// TwinCAT 3 PLC project TwinCAT_OpenFramework_IO_Models
// Title: TwinCAT Open Framework IO Models
// Company: Oleksandr Tiutyk FOP
// Author: Oleksandr Tiutyk
// ProjectVersion: 1.0.13.0
// Description: Beckhoff I/O (input/output) models: different terminal models
// ProgramVersion: 3.1.4026.28
// project tree:
//   AnalogIO/Inputs/ ANALOG_INPUT_DINT_CHANNEL.TcDUT, ANALOG_INPUT_REAL_CHANNEL.TcDUT, ANALOG_INPUT_INT_CHANNEL.TcDUT, RTD_INPUT_CHANNEL.TcDUT, THERMOCOUPLE_INPUT_CHANNEL.TcDUT
//   AnalogIO/Inputs/EL3002/ EL3002.TcDUT, EL3002_EX.TcDUT
//   AnalogIO/Inputs/EL3004/ EL3004.TcDUT, EL3004_EX.TcDUT
//   AnalogIO/Inputs/EL3008/ EL3008.TcDUT, EL3008_EX.TcDUT
//   AnalogIO/Inputs/EL3078/ EL3078.TcDUT, EL3078_EX.TcDUT
//   AnalogIO/Inputs/EL3001/ EL3001.TcDUT, EL3001_EX.TcDUT
//   AnalogIO/Outputs/EL4001/ EL4001.TcDUT, EL4001_EX.TcDUT
//   AnalogIO/Outputs/EL4002/ EL4002.TcDUT, EL4002_EX.TcDUT
//   AnalogIO/Outputs/EL4004/ EL4004.TcDUT, EL4004_EX.TcDUT
//   AnalogIO/Outputs/EL4008/ EL4008.TcDUT, EL4008_EX.TcDUT
//   DigitalIO/Inputs/EL1002/ EL1002.TcDUT, EL1002_EX.TcDUT
//   DigitalIO/Inputs/EL1004/ EL1004.TcDUT, EL1004_EX.TcDUT
//   DigitalIO/Inputs/EL1018/ EL1018_EX.TcDUT, EL1018.TcDUT
//   DigitalIO/Inputs/EL1809/ EL1809.TcDUT, EL1809_EX.TcDUT
//   DigitalIO/Outputs/EL2008/ EL2008.TcDUT, EL2008_EX.TcDUT
//   DigitalIO/Outputs/EL2002/ EL2002.TcDUT, EL2002_EX.TcDUT
//   DigitalIO/Outputs/EL2004/ EL2004.TcDUT, EL2004_EX.TcDUT
//   DigitalIO/Outputs/EL2409/ EL2409.TcDUT, EL2409_EX.TcDUT
//   Internal/ CurrentNamespace.TcPOU, NamespaceExtractor.TcPOU
//   Serial/EL6022/ EL6022.TcDUT, EL6022_CHANNEL.TcDUT, EL6022_EX.TcDUT
//   Serial/ EL6xxx22ByteInData.TcDUT, EL6xxx22ByteOutData.TcDUT
//   AnalogIO/Inputs/EL3201/ EL3201.TcDUT, EL3201_EX.TcDUT
//   AnalogIO/Inputs/EL3202/ EL3202.TcDUT, EL3202_EX.TcDUT
//   AnalogIO/Inputs/EL3204/ EL3204.TcDUT, EL3204_EX.TcDUT
//   AnalogIO/Inputs/EL3208/ EL3208.TcDUT, EL3208_EX.TcDUT
//   AnalogIO/Inputs/EL3311/ EL3311.TcDUT, EL3311_EX.TcDUT
//   AnalogIO/Inputs/EL3312/ EL3312.TcDUT, EL3312_EX.TcDUT
//   AnalogIO/Inputs/EL3314/ EL3314.TcDUT, EL3314_EX.TcDUT
//   AnalogIO/Inputs/EL3318/ EL3318.TcDUT, EL3318_EX.TcDUT
//   DigitalIO/Inputs/EL1008/ EL1008.TcDUT, EL1008_EX.TcDUT
//   DigitalIO/Outputs/EL2809/ EL2809.TcDUT, EL2809_EX.TcDUT
//   DigitalIO/Outputs/EL2622/ EL2622.TcDUT, EL2622_EX.TcDUT
//   DigitalIO/Outputs/EL2624/ EL2624.TcDUT, EL2624_EX.TcDUT
//   Serial/EL6001/ EL6001.TcDUT, EL6001_CHANNEL.TcDUT, EL6001_EX.TcDUT
//   Serial/EL6002/ EL6002.TcDUT, EL6002_CHANNEL.TcDUT, EL6002_EX.TcDUT
//   Serial/EL6021/ EL6021.TcDUT, EL6021_CHANNEL.TcDUT, EL6021_EX.TcDUT
//   Counters/ COUNTER_INPUT_CHANNEL.TcDUT, COUNTER_OUTPUT_CHANNEL.TcDUT, COUNTER_CHANNEL.TcDUT
//   Counters/EL1502/ EL1502.TcDUT, EL1502_EX.TcDUT
//   Counters/EL1512/ EL1512.TcDUT, EL1512_EX.TcDUT
//   Encoders/ INCREMENTAL_ENCODER_INPUT_CHANNEL.TcDUT, INCREMENTAL_ENCODER_OUTPUT_CHANNEL.TcDUT, INCREMENTAL_ENCODER_CHANNEL.TcDUT, INCREMENTAL_ENCODER_COUNTER_INPUT_CHANNEL.TcDUT, INCREMENTAL_ENCODER_COUNTER_CHANNEL.TcDUT, SSI_ENCODER_CHANNEL.TcDUT
//   Encoders/EL5101/ EL5101.TcDUT, EL5101_EX.TcDUT
//   Encoders/EL5151/ EL5151.TcDUT, EL5151_EX.TcDUT
//   Encoders/EL5152/ EL5152.TcDUT, EL5152_EX.TcDUT
//   Encoders/EL5001/ EL5001.TcDUT, EL5001_EX.TcDUT
//   Encoders/EL5002/ EL5002.TcDUT, EL5002_EX.TcDUT
//   PWM/ PWM_OUTPUT_CHANNEL.TcDUT, PULSE_TRAIN_INPUT_CHANNEL.TcDUT, PULSE_TRAIN_OUTPUT_CHANNEL.TcDUT, PULSE_TRAIN_CHANNEL.TcDUT
//   PWM/EL2502/ EL2502.TcDUT, EL2502_EX.TcDUT
//   PWM/EL2521/ EL2521.TcDUT, EL2521_EX.TcDUT
//   Version/ Global_Version.TcGVL
//   AnalogIO/Inputs/EL3051/ EL3051.TcDUT, EL3051_EX.TcDUT
//   AnalogIO/Inputs/EL3052/ EL3052.TcDUT, EL3052_EX.TcDUT
//   AnalogIO/Inputs/EL3054/ EL3054.TcDUT, EL3054_EX.TcDUT
//   AnalogIO/Inputs/EL3058/ EL3058.TcDUT, EL3058_EX.TcDUT
//   AnalogIO/Inputs/EL3102/ EL3102.TcDUT, EL3102_EX.TcDUT
//   AnalogIO/Inputs/EL3104/ EL3104.TcDUT, EL3104_EX.TcDUT
//   AnalogIO/Inputs/EL3122/ EL3122.TcDUT, EL3122_EX.TcDUT
//   AnalogIO/Inputs/EL3124/ EL3124.TcDUT, EL3124_EX.TcDUT
//   AnalogIO/Outputs/EL4021/ EL4021.TcDUT, EL4021_EX.TcDUT
//   AnalogIO/Outputs/EL4022/ EL4022.TcDUT, EL4022_EX.TcDUT
//   AnalogIO/Outputs/EL4024/ EL4024.TcDUT, EL4024_EX.TcDUT
//   AnalogIO/Outputs/EL4028/ EL4028.TcDUT, EL4028_EX.TcDUT
//   AnalogIO/Outputs/EL4102/ EL4102.TcDUT, EL4102_EX.TcDUT
//   AnalogIO/Outputs/EL4104/ EL4104.TcDUT, EL4104_EX.TcDUT
//   AnalogIO/Outputs/EL4132/ EL4132.TcDUT, EL4132_EX.TcDUT
//   AnalogIO/Outputs/EL4134/ EL4134.TcDUT, EL4134_EX.TcDUT
//   AnalogIO/Outputs/EL4122/ EL4122.TcDUT, EL4122_EX.TcDUT
//   AnalogIO/Outputs/EL4124/ EL4124.TcDUT, EL4124_EX.TcDUT
//   Weighing/ STRAIN_GAUGE_INPUT_CHANNEL.TcDUT, STRAIN_GAUGE_OUTPUT_CHANNEL.TcDUT, STRAIN_GAUGE_CHANNEL.TcDUT
//   Weighing/EL3356/ EL3356.TcDUT, EL3356_EX.TcDUT
//   Weighing/EL3356_0010/ EL3356_0010.TcDUT, EL3356_0010_EX.TcDUT
//   PowerMeasurement/ POWER_MEASUREMENT_INPUT_CHANNEL.TcDUT, POWER_MEASUREMENT_OUTPUT_CHANNEL.TcDUT, POWER_MEASUREMENT_CHANNEL.TcDUT, POWER_MEASUREMENT_AUXILIARY_INPUT_CHANNEL.TcDUT, POWER_MEASUREMENT_AUXILIARY_OUTPUT_CHANNEL.TcDUT, POWER_MEASUREMENT_AUXILIARY_CHANNEL.TcDUT
//   PowerMeasurement/EL3403/ EL3403.TcDUT, EL3403_INPUT_CHANNEL.TcDUT, EL3403_CHANNEL.TcDUT, EL3403_EX.TcDUT
//   PowerMeasurement/EL3413/ EL3413.TcDUT, EL3413_EX.TcDUT
//   PowerMeasurement/EL3433/ EL3433.TcDUT, EL3433_EX.TcDUT
//   DigitalIO/Inputs/EP1008_0001/ EP1008_0001.TcDUT, EP1008_0001_EX.TcDUT
//   DigitalIO/Inputs/EP1008_0002/ EP1008_0002.TcDUT, EP1008_0002_EX.TcDUT
//   DigitalIO/Inputs/EP1018_0001/ EP1018_0001.TcDUT, EP1018_0001_EX.TcDUT
//   DigitalIO/Inputs/EP1809_0021/ EP1809_0021.TcDUT, EP1809_0021_EX.TcDUT
//   DigitalIO/Outputs/EP2008_0001/ EP2008_0001.TcDUT, EP2008_0001_EX.TcDUT
//   DigitalIO/Outputs/EP2008_0002/ EP2008_0002.TcDUT, EP2008_0002_EX.TcDUT
//   DigitalIO/Outputs/EP2809_0021/ EP2809_0021.TcDUT, EP2809_0021_EX.TcDUT
//   DigitalIO/Outputs/EP2624_0002/ EP2624_0002.TcDUT, EP2624_0002_EX.TcDUT
//   AnalogIO/Inputs/EP3174_0002/ EP3174_0002.TcDUT, EP3174_0002_EX.TcDUT
//   AnalogIO/Outputs/EP4174_0002/ EP4174_0002.TcDUT, EP4174_0002_EX.TcDUT
//   Serial/EP6001_0002/ EP6001_0002.TcDUT, EP6001_0002_EX.TcDUT
//   Serial/EP6002_0002/ EP6002_0002.TcDUT, EP6002_0002_EX.TcDUT
// (motion and I/O tree: see PLC project twincat_openframework_core)
// real-time tasks:
//   TASK PlcTask: cycle T#10ms, priority 20, ADS port 350
//   TASK TestTask: cycle T#10ms, priority 1, ADS port 351
//   TASK RunnerTestTask: cycle T#10ms, priority 2, ADS port 354
//   TASK HowToTask: cycle T#10ms, priority 22, ADS port 353
// variable links:

// ---- AnalogIO/Inputs/ANALOG_INPUT_DINT_CHANNEL.TcDUT
(*
SPDX-FileCopyrightText: © 2026 Oleksandr Tiutyk <trofimich@gmail.com>
SPDX-License-Identifier: MIT
License: https://opensource.org/license/mit
*)

(*!
<summary>
Beckhoff 32-bit analog input channel process image.
</summary>
<description>
Encapsulates a 16-bit status word and a 32-bit signed double-integer raw value '%I*' for high-resolution
analog input channels.
When used for I/O, link located fields or their containing buffers to the matching selected PDOs.
The record is not a packed wire buffer; compiler padding is not part of the device specification.
Unlinked/default values do not prove valid I/O. The caller evaluates bus/channel validity before use.
Use one owner task per instance and externally synchronize other access; multi-field snapshots are not atomic.
Copies store data without creating hardware links. Keep borrowed field references valid while consumers are bound.
This passive record performs no validation, synchronization, configuration or protocol advancement.
Select standard status-plus-value PDOs matching the declared Value type; compact value-only PDOs
are outside this model. Configure electrical range and scaling separately on the device.
</description>
*)
TYPE ANALOG_INPUT_DINT_CHANNEL :
STRUCT
	Status AT %I* : WORD;
	Value AT %I* : DINT;
END_STRUCT
END_TYPE

// ---- AnalogIO/Inputs/ANALOG_INPUT_REAL_CHANNEL.TcDUT
(*
SPDX-FileCopyrightText: © 2026 Oleksandr Tiutyk <trofimich@gmail.com>
SPDX-License-Identifier: MIT
License: https://opensource.org/license/mit
*)

(*!
<summary>
Beckhoff floating-point analog input channel process image.
</summary>
<description>
Encapsulates a 16-bit status word and a 32-bit single-precision REAL process value '%I*' for multi-range
analog input channels.
When used for I/O, link located fields or their containing buffers to the matching selected PDOs.
The record is not a packed wire buffer; compiler padding is not part of the device specification.
Unlinked/default values do not prove valid I/O. The caller evaluates bus/channel validity before use.
Use one owner task per instance and externally synchronize other access; multi-field snapshots are not atomic.
Copies store data without creating hardware links. Keep borrowed field references valid while consumers are bound.
This passive record performs no validation, synchronization, configuration or protocol advancement.
Select standard status-plus-value PDOs matching the declared Value type; compact value-only PDOs
are outside this model. Configure electrical range and scaling separately on the device.
</description>
*)
TYPE ANALOG_INPUT_REAL_CHANNEL :
STRUCT
	Status AT %I* : WORD;
	Value AT %I* : REAL;
END_STRUCT
END_TYPE

// ---- AnalogIO/Inputs/ANALOG_INPUT_INT_CHANNEL.TcDUT
(*
SPDX-FileCopyrightText: © 2026 Oleksandr Tiutyk <trofimich@gmail.com>
SPDX-License-Identifier: MIT
License: https://opensource.org/license/mit
*)

(*!
<summary>
Beckhoff 16-bit analog input channel process image.
</summary>
<description>
Encapsulates a 16-bit status word and a 16-bit signed integer raw value '%I*' for standard analog input
channels.
When used for I/O, link located fields or their containing buffers to the matching selected PDOs.
The record is not a packed wire buffer; compiler padding is not part of the device specification.
Unlinked/default values do not prove valid I/O. The caller evaluates bus/channel validity before use.
Use one owner task per instance and externally synchronize other access; multi-field snapshots are not atomic.
Copies store data without creating hardware links. Keep borrowed field references valid while consumers are bound.
This passive record performs no validation, synchronization, configuration or protocol advancement.
Select standard status-plus-value PDOs matching the declared Value type; compact value-only PDOs
are outside this model. Configure electrical range and scaling separately on the device.
</description>
*)
TYPE ANALOG_INPUT_INT_CHANNEL :
STRUCT
	Status AT %I* : WORD;
	Value AT %I* : INT;
END_STRUCT
END_TYPE

// ---- AnalogIO/Inputs/EL3002/EL3002.TcDUT
(*
SPDX-FileCopyrightText: © 2026 Oleksandr Tiutyk <trofimich@gmail.com>
SPDX-License-Identifier: MIT
License: https://opensource.org/license/mit
*)

(*!
<summary>
Beckhoff EL3002: 2-channel analog input terminal (-10 V .. +10 V, 12-bit).
</summary>
<description>
Process image mapping structure for the EL3002 EtherCAT terminal with 2 analog input channels.
When used for I/O, link located fields or their containing buffers to the matching selected PDOs.
The record is not a packed wire buffer; compiler padding is not part of the device specification.
Unlinked/default values do not prove valid I/O. The caller evaluates bus/channel validity before use.
Use one owner task per instance and externally synchronize other access; multi-field snapshots are not atomic.
Copies store data without creating hardware links. Keep borrowed field references valid while consumers are bound.
This passive record performs no validation, synchronization, configuration or protocol advancement.
Select standard status-plus-value PDOs matching the declared Value type; compact value-only PDOs
are outside this model. Configure electrical range and scaling separately on the device.
</description>
*)
TYPE EL3002 :
STRUCT
	Ch1 : ANALOG_INPUT_INT_CHANNEL;
	Ch2 : ANALOG_INPUT_INT_CHANNEL;
END_STRUCT
END_TYPE

// ---- AnalogIO/Inputs/EL3002/EL3002_EX.TcDUT
(*
SPDX-FileCopyrightText: © 2026 Oleksandr Tiutyk <trofimich@gmail.com>
SPDX-License-Identifier: MIT
License: https://opensource.org/license/mit
*)

(*!
<summary>
Beckhoff EL3002_EX: Extended 2-channel analog input terminal with diagnostics.
</summary>
<description>
Extends EL3002 with EtherCAT Working Counter, slave state, and CoE mailbox ADS address diagnostics.
When used for I/O, link located fields or their containing buffers to the matching selected PDOs.
The record is not a packed wire buffer; compiler padding is not part of the device specification.
Unlinked/default values do not prove valid I/O. The caller evaluates bus/channel validity before use.
Use one owner task per instance and externally synchronize other access; multi-field snapshots are not atomic.
Copies store data without creating hardware links. Keep borrowed field references valid while consumers are bound.
This passive record performs no validation, synchronization, configuration or protocol advancement.
WcState=TRUE means process-data exchange is invalid. State is acyclic EtherCAT/link information,
not proof of current measurement validity. Link diagnostics to the matching slave InfoData entries.
The selected PDO representation is documented by the base terminal model.
InputToggle signals an input update by changing state; TRUE alone does not mean fresh data.
AdsAddr is acyclic mailbox addressing information, not a measurement-validity indicator.
Select standard status-plus-value PDOs matching the declared Value type; compact value-only PDOs
are outside this model. Configure electrical range and scaling separately on the device.
</description>
*)
TYPE EL3002_EX EXTENDS EL3002 :
STRUCT
	WcState AT %I* : BOOL;
	InputToggle AT %I* : BOOL;
	State AT %I* : UINT;
	AdsAddr AT %I* : Global.AMSADDR;
END_STRUCT
END_TYPE

// ---- AnalogIO/Inputs/EL3004/EL3004.TcDUT
(*
SPDX-FileCopyrightText: © 2026 Oleksandr Tiutyk <trofimich@gmail.com>
SPDX-License-Identifier: MIT
License: https://opensource.org/license/mit
*)

(*!
<summary>
Beckhoff EL3004: 4-channel analog input terminal (-10 V .. +10 V, 12-bit).
</summary>
<description>
Process image mapping structure for the EL3004 EtherCAT terminal with 4 analog input channels.
When used for I/O, link located fields or their containing buffers to the matching selected PDOs.
The record is not a packed wire buffer; compiler padding is not part of the device specification.
Unlinked/default values do not prove valid I/O. The caller evaluates bus/channel validity before use.
Use one owner task per instance and externally synchronize other access; multi-field snapshots are not atomic.
Copies store data without creating hardware links. Keep borrowed field references valid while consumers are bound.
This passive record performs no validation, synchronization, configuration or protocol advancement.
Select standard status-plus-value PDOs matching the declared Value type; compact value-only PDOs
are outside this model. Configure electrical range and scaling separately on the device.
</description>
*)
TYPE EL3004 :
STRUCT
	Ch1 : ANALOG_INPUT_INT_CHANNEL;
	Ch2 : ANALOG_INPUT_INT_CHANNEL;
	Ch3 : ANALOG_INPUT_INT_CHANNEL;
	Ch4 : ANALOG_INPUT_INT_CHANNEL;
END_STRUCT
END_TYPE

// ---- AnalogIO/Inputs/EL3004/EL3004_EX.TcDUT
(*
SPDX-FileCopyrightText: © 2026 Oleksandr Tiutyk <trofimich@gmail.com>
SPDX-License-Identifier: MIT
License: https://opensource.org/license/mit
*)

(*!
<summary>
Beckhoff EL3004_EX: Extended 4-channel analog input terminal with diagnostics.
</summary>
<description>
Extends EL3004 with EtherCAT Working Counter, slave state, and CoE mailbox ADS address diagnostics.
When used for I/O, link located fields or their containing buffers to the matching selected PDOs.
The record is not a packed wire buffer; compiler padding is not part of the device specification.
Unlinked/default values do not prove valid I/O. The caller evaluates bus/channel validity before use.
Use one owner task per instance and externally synchronize other access; multi-field snapshots are not atomic.
Copies store data without creating hardware links. Keep borrowed field references valid while consumers are bound.
This passive record performs no validation, synchronization, configuration or protocol advancement.
WcState=TRUE means process-data exchange is invalid. State is acyclic EtherCAT/link information,
not proof of current measurement validity. Link diagnostics to the matching slave InfoData entries.
The selected PDO representation is documented by the base terminal model.
InputToggle signals an input update by changing state; TRUE alone does not mean fresh data.
AdsAddr is acyclic mailbox addressing information, not a measurement-validity indicator.
Select standard status-plus-value PDOs matching the declared Value type; compact value-only PDOs
are outside this model. Configure electrical range and scaling separately on the device.
</description>
*)
TYPE EL3004_EX EXTENDS EL3004 :
STRUCT
	WcState AT %I* : BOOL;
	InputToggle AT %I* : BOOL;
	State AT %I* : UINT;
	AdsAddr AT %I* : Global.AMSADDR;
END_STRUCT
END_TYPE

// ---- AnalogIO/Inputs/EL3008/EL3008.TcDUT
(*
SPDX-FileCopyrightText: © 2026 Oleksandr Tiutyk <trofimich@gmail.com>
SPDX-License-Identifier: MIT
License: https://opensource.org/license/mit
*)

(*!
<summary>
Beckhoff EL3008: 8-channel analog input terminal (-10 V .. +10 V, 12-bit).
</summary>
<description>
Process image mapping structure for the EL3008 EtherCAT terminal with 8 analog input channels.
When used for I/O, link located fields or their containing buffers to the matching selected PDOs.
The record is not a packed wire buffer; compiler padding is not part of the device specification.
Unlinked/default values do not prove valid I/O. The caller evaluates bus/channel validity before use.
Use one owner task per instance and externally synchronize other access; multi-field snapshots are not atomic.
Copies store data without creating hardware links. Keep borrowed field references valid while consumers are bound.
This passive record performs no validation, synchronization, configuration or protocol advancement.
Select standard status-plus-value PDOs matching the declared Value type; compact value-only PDOs
are outside this model. Configure electrical range and scaling separately on the device.
</description>
*)
TYPE EL3008 :
STRUCT
	Ch1 : ANALOG_INPUT_INT_CHANNEL;
	Ch2 : ANALOG_INPUT_INT_CHANNEL;
	Ch3 : ANALOG_INPUT_INT_CHANNEL;
	Ch4 : ANALOG_INPUT_INT_CHANNEL;
	Ch5 : ANALOG_INPUT_INT_CHANNEL;
	Ch6 : ANALOG_INPUT_INT_CHANNEL;
	Ch7 : ANALOG_INPUT_INT_CHANNEL;
	Ch8 : ANALOG_INPUT_INT_CHANNEL;
END_STRUCT
END_TYPE

// ---- AnalogIO/Inputs/EL3008/EL3008_EX.TcDUT
(*
SPDX-FileCopyrightText: © 2026 Oleksandr Tiutyk <trofimich@gmail.com>
SPDX-License-Identifier: MIT
License: https://opensource.org/license/mit
*)

(*!
<summary>
Beckhoff EL3008_EX: Extended 8-channel analog input terminal with diagnostics.
</summary>
<description>
Extends EL3008 with EtherCAT Working Counter, slave state, and CoE mailbox ADS address diagnostics.
When used for I/O, link located fields or their containing buffers to the matching selected PDOs.
The record is not a packed wire buffer; compiler padding is not part of the device specification.
Unlinked/default values do not prove valid I/O. The caller evaluates bus/channel validity before use.
Use one owner task per instance and externally synchronize other access; multi-field snapshots are not atomic.
Copies store data without creating hardware links. Keep borrowed field references valid while consumers are bound.
This passive record performs no validation, synchronization, configuration or protocol advancement.
WcState=TRUE means process-data exchange is invalid. State is acyclic EtherCAT/link information,
not proof of current measurement validity. Link diagnostics to the matching slave InfoData entries.
The selected PDO representation is documented by the base terminal model.
InputToggle signals an input update by changing state; TRUE alone does not mean fresh data.
AdsAddr is acyclic mailbox addressing information, not a measurement-validity indicator.
Select standard status-plus-value PDOs matching the declared Value type; compact value-only PDOs
are outside this model. Configure electrical range and scaling separately on the device.
</description>
*)
TYPE EL3008_EX EXTENDS EL3008 :
STRUCT
	WcState AT %I* : BOOL;
	InputToggle AT %I* : BOOL;
	State AT %I* : UINT;
	AdsAddr AT %I* : Global.AMSADDR;
END_STRUCT
END_TYPE

// ---- AnalogIO/Inputs/EL3078/EL3078.TcDUT
(*
SPDX-FileCopyrightText: © 2026 Oleksandr Tiutyk <trofimich@gmail.com>
SPDX-License-Identifier: MIT
License: https://opensource.org/license/mit
*)

(*!
<summary>
Beckhoff EL3078: 8-channel multi-range analog input terminal (REAL values).
</summary>
<description>
Process image mapping structure for the EL3078 EtherCAT terminal with 8 multi-range analog input channels
outputting REAL floating-point values.
Requires AI Standard (Real32) TxPDOs 0x1A10, 0x1A12, 0x1A14, 0x1A16, 0x1A18, 0x1A1A, 0x1A1C and 0x1A1E.
Value entries at 0x60n0:13 are REAL32; INT16 and compact assignments are outside this model.
When used for I/O, link located fields or their containing buffers to the matching selected PDOs.
The record is not a packed wire buffer; compiler padding is not part of the device specification.
Unlinked/default values do not prove valid I/O. The caller evaluates bus/channel validity before use.
Use one owner task per instance and externally synchronize other access; multi-field snapshots are not atomic.
Copies store data without creating hardware links. Keep borrowed field references valid while consumers are bound.
This passive record performs no validation, synchronization, configuration or protocol advancement.
Select standard status-plus-value PDOs matching the declared Value type; compact value-only PDOs
are outside this model. Configure electrical range and scaling separately on the device.
</description>
*)
TYPE EL3078 :
STRUCT
	Ch1 : ANALOG_INPUT_REAL_CHANNEL;
	Ch2 : ANALOG_INPUT_REAL_CHANNEL;
	Ch3 : ANALOG_INPUT_REAL_CHANNEL;
	Ch4 : ANALOG_INPUT_REAL_CHANNEL;
	Ch5 : ANALOG_INPUT_REAL_CHANNEL;
	Ch6 : ANALOG_INPUT_REAL_CHANNEL;
	Ch7 : ANALOG_INPUT_REAL_CHANNEL;
	Ch8 : ANALOG_INPUT_REAL_CHANNEL;
END_STRUCT
END_TYPE

// ---- AnalogIO/Inputs/EL3078/EL3078_EX.TcDUT
(*
SPDX-FileCopyrightText: © 2026 Oleksandr Tiutyk <trofimich@gmail.com>
SPDX-License-Identifier: MIT
License: https://opensource.org/license/mit
*)

(*!
<summary>
Beckhoff EL3078_EX: Extended 8-channel multi-range analog input terminal with diagnostics.
</summary>
<description>
Extends EL3078 with EtherCAT Working Counter, slave state, and CoE mailbox ADS address diagnostics.
When used for I/O, link located fields or their containing buffers to the matching selected PDOs.
The record is not a packed wire buffer; compiler padding is not part of the device specification.
Unlinked/default values do not prove valid I/O. The caller evaluates bus/channel validity before use.
Use one owner task per instance and externally synchronize other access; multi-field snapshots are not atomic.
Copies store data without creating hardware links. Keep borrowed field references valid while consumers are bound.
This passive record performs no validation, synchronization, configuration or protocol advancement.
WcState=TRUE means process-data exchange is invalid. State is acyclic EtherCAT/link information,
not proof of current measurement validity. Link diagnostics to the matching slave InfoData entries.
The selected PDO representation is documented by the base terminal model.
InputToggle signals an input update by changing state; TRUE alone does not mean fresh data.
AdsAddr is acyclic mailbox addressing information, not a measurement-validity indicator.
Select standard status-plus-value PDOs matching the declared Value type; compact value-only PDOs
are outside this model. Configure electrical range and scaling separately on the device.
</description>
*)
TYPE EL3078_EX EXTENDS EL3078 :
STRUCT
	WcState AT %I* : BOOL;
	InputToggle AT %I* : BOOL;
	State AT %I* : UINT;
	AdsAddr AT %I* : Global.AMSADDR;
END_STRUCT
END_TYPE

// ---- AnalogIO/Inputs/EL3001/EL3001.TcDUT
(*
SPDX-FileCopyrightText: © 2026 Oleksandr Tiutyk <trofimich@gmail.com>
SPDX-License-Identifier: MIT
License: https://opensource.org/license/mit
*)

(*!
<summary>
Beckhoff EL3001: 1-channel analog input terminal (-10 V .. +10 V, 12-bit).
</summary>
<description>
Process image mapping structure for the EL3001 EtherCAT terminal with 1 analog input channel.
When used for I/O, link located fields or their containing buffers to the matching selected PDOs.
The record is not a packed wire buffer; compiler padding is not part of the device specification.
Unlinked/default values do not prove valid I/O. The caller evaluates bus/channel validity before use.
Use one owner task per instance and externally synchronize other access; multi-field snapshots are not atomic.
Copies store data without creating hardware links. Keep borrowed field references valid while consumers are bound.
This passive record performs no validation, synchronization, configuration or protocol advancement.
Select standard status-plus-value PDOs matching the declared Value type; compact value-only PDOs
are outside this model. Configure electrical range and scaling separately on the device.
</description>
*)
TYPE EL3001 :
STRUCT
	Ch1 : ANALOG_INPUT_INT_CHANNEL;
END_STRUCT
END_TYPE

// ---- AnalogIO/Inputs/EL3001/EL3001_EX.TcDUT
(*
SPDX-FileCopyrightText: © 2026 Oleksandr Tiutyk <trofimich@gmail.com>
SPDX-License-Identifier: MIT
License: https://opensource.org/license/mit
*)

(*!
<summary>
Beckhoff EL3001_EX: Extended 1-channel analog input terminal with diagnostics.
</summary>
<description>
Extends EL3001 with EtherCAT Working Counter, slave state, and CoE mailbox ADS address diagnostics.
When used for I/O, link located fields or their containing buffers to the matching selected PDOs.
The record is not a packed wire buffer; compiler padding is not part of the device specification.
Unlinked/default values do not prove valid I/O. The caller evaluates bus/channel validity before use.
Use one owner task per instance and externally synchronize other access; multi-field snapshots are not atomic.
Copies store data without creating hardware links. Keep borrowed field references valid while consumers are bound.
This passive record performs no validation, synchronization, configuration or protocol advancement.
WcState=TRUE means process-data exchange is invalid. State is acyclic EtherCAT/link information,
not proof of current measurement validity. Link diagnostics to the matching slave InfoData entries.
The selected PDO representation is documented by the base terminal model.
InputToggle signals an input update by changing state; TRUE alone does not mean fresh data.
AdsAddr is acyclic mailbox addressing information, not a measurement-validity indicator.
Select standard status-plus-value PDOs matching the declared Value type; compact value-only PDOs
are outside this model. Configure electrical range and scaling separately on the device.
</description>
*)
TYPE EL3001_EX EXTENDS EL3001 :
STRUCT
	WcState AT %I* : BOOL;
	InputToggle AT %I* : BOOL;
	State AT %I* : UINT;
	AdsAddr AT %I* : Global.AMSADDR;
END_STRUCT
END_TYPE

// ---- AnalogIO/Outputs/EL4001/EL4001.TcDUT
(*
SPDX-FileCopyrightText: © 2026 Oleksandr Tiutyk <trofimich@gmail.com>
SPDX-License-Identifier: MIT
License: https://opensource.org/license/mit
*)

(*!
<summary>
Beckhoff EL4001: 1-channel analog output terminal (0 .. 10 V, 12-bit).
</summary>
<description>
Process image mapping structure for the EL4001 EtherCAT terminal with 1 analog output channel (0 .. 10 V,
12-bit).
When used for I/O, link located fields or their containing buffers to the matching selected PDOs.
The record is not a packed wire buffer; compiler padding is not part of the device specification.
Unlinked/default values do not prove valid I/O. The caller evaluates bus/channel validity before use.
Use one owner task per instance and externally synchronize other access; multi-field snapshots are not atomic.
Copies store data without creating hardware links. Keep borrowed field references valid while consumers are bound.
This passive record performs no validation, synchronization, configuration or protocol advancement.
Channels hold raw INT16 output commands; configure electrical range and presentation before use.
</description>
*)
TYPE EL4001 :
STRUCT
	Ch1 AT %Q* : INT;
END_STRUCT
END_TYPE

// ---- AnalogIO/Outputs/EL4001/EL4001_EX.TcDUT
(*
SPDX-FileCopyrightText: © 2026 Oleksandr Tiutyk <trofimich@gmail.com>
SPDX-License-Identifier: MIT
License: https://opensource.org/license/mit
*)

(*!
<summary>
Beckhoff EL4001_EX: Extended 1-channel analog output terminal with diagnostics.
</summary>
<description>
Extends EL4001 with EtherCAT Working Counter and slave state diagnostics.
When used for I/O, link located fields or their containing buffers to the matching selected PDOs.
The record is not a packed wire buffer; compiler padding is not part of the device specification.
Unlinked/default values do not prove valid I/O. The caller evaluates bus/channel validity before use.
Use one owner task per instance and externally synchronize other access; multi-field snapshots are not atomic.
Copies store data without creating hardware links. Keep borrowed field references valid while consumers are bound.
This passive record performs no validation, synchronization, configuration or protocol advancement.
WcState=TRUE means process-data exchange is invalid. State is acyclic EtherCAT/link information,
not proof of current measurement validity. Link diagnostics to the matching slave InfoData entries.
The selected PDO representation is documented by the base terminal model.
AdsAddr is acyclic mailbox addressing information, not a measurement-validity indicator.
Channels hold raw INT16 output commands; configure electrical range and presentation before use.
</description>
*)
TYPE EL4001_EX EXTENDS EL4001 :
STRUCT
	WcState AT %I* : BOOL;
	State AT %I* : UINT;
	AdsAddr AT %I* : Global.AMSADDR;
END_STRUCT
END_TYPE

// ---- AnalogIO/Outputs/EL4002/EL4002.TcDUT
(*
SPDX-FileCopyrightText: © 2026 Oleksandr Tiutyk <trofimich@gmail.com>
SPDX-License-Identifier: MIT
License: https://opensource.org/license/mit
*)

(*!
<summary>
Beckhoff EL4002: 2-channel analog output terminal (0 .. 10 V, 12-bit).
</summary>
<description>
Process image mapping structure for the EL4002 EtherCAT terminal with 2 analog output channels (0 .. 10 V,
12-bit).
When used for I/O, link located fields or their containing buffers to the matching selected PDOs.
The record is not a packed wire buffer; compiler padding is not part of the device specification.
Unlinked/default values do not prove valid I/O. The caller evaluates bus/channel validity before use.
Use one owner task per instance and externally synchronize other access; multi-field snapshots are not atomic.
Copies store data without creating hardware links. Keep borrowed field references valid while consumers are bound.
This passive record performs no validation, synchronization, configuration or protocol advancement.
Channels hold raw INT16 output commands; configure electrical range and presentation before use.
</description>
*)
TYPE EL4002 :
STRUCT
	Ch1 AT %Q* : INT;
	Ch2 AT %Q* : INT;
END_STRUCT
END_TYPE

// ---- AnalogIO/Outputs/EL4002/EL4002_EX.TcDUT
(*
SPDX-FileCopyrightText: © 2026 Oleksandr Tiutyk <trofimich@gmail.com>
SPDX-License-Identifier: MIT
License: https://opensource.org/license/mit
*)

(*!
<summary>
Beckhoff EL4002_EX: Extended 2-channel analog output terminal with diagnostics.
</summary>
<description>
Extends EL4002 with EtherCAT Working Counter and slave state diagnostics.
When used for I/O, link located fields or their containing buffers to the matching selected PDOs.
The record is not a packed wire buffer; compiler padding is not part of the device specification.
Unlinked/default values do not prove valid I/O. The caller evaluates bus/channel validity before use.
Use one owner task per instance and externally synchronize other access; multi-field snapshots are not atomic.
Copies store data without creating hardware links. Keep borrowed field references valid while consumers are bound.
This passive record performs no validation, synchronization, configuration or protocol advancement.
WcState=TRUE means process-data exchange is invalid. State is acyclic EtherCAT/link information,
not proof of current measurement validity. Link diagnostics to the matching slave InfoData entries.
The selected PDO representation is documented by the base terminal model.
AdsAddr is acyclic mailbox addressing information, not a measurement-validity indicator.
Channels hold raw INT16 output commands; configure electrical range and presentation before use.
</description>
*)
TYPE EL4002_EX EXTENDS EL4002 :
STRUCT
	WcState AT %I* : BOOL;
	State AT %I* : UINT;
	AdsAddr AT %I* : Global.AMSADDR;
END_STRUCT
END_TYPE

// ---- AnalogIO/Outputs/EL4004/EL4004.TcDUT
(*
SPDX-FileCopyrightText: © 2026 Oleksandr Tiutyk <trofimich@gmail.com>
SPDX-License-Identifier: MIT
License: https://opensource.org/license/mit
*)

(*!
<summary>
Beckhoff EL4004: 4-channel analog output terminal (0 .. 10 V, 12-bit).
</summary>
<description>
Process image mapping structure for the EL4004 EtherCAT terminal with 4 analog output channels (0 .. 10 V,
12-bit).
When used for I/O, link located fields or their containing buffers to the matching selected PDOs.
The record is not a packed wire buffer; compiler padding is not part of the device specification.
Unlinked/default values do not prove valid I/O. The caller evaluates bus/channel validity before use.
Use one owner task per instance and externally synchronize other access; multi-field snapshots are not atomic.
Copies store data without creating hardware links. Keep borrowed field references valid while consumers are bound.
This passive record performs no validation, synchronization, configuration or protocol advancement.
Channels hold raw INT16 output commands; configure electrical range and presentation before use.
</description>
*)
TYPE EL4004 :
STRUCT
	Ch1 AT %Q* : INT;
	Ch2 AT %Q* : INT;
	Ch3 AT %Q* : INT;
	Ch4 AT %Q* : INT;
END_STRUCT
END_TYPE

// ---- AnalogIO/Outputs/EL4004/EL4004_EX.TcDUT
(*
SPDX-FileCopyrightText: © 2026 Oleksandr Tiutyk <trofimich@gmail.com>
SPDX-License-Identifier: MIT
License: https://opensource.org/license/mit
*)

(*!
<summary>
Beckhoff EL4004_EX: Extended 4-channel analog output terminal with diagnostics.
</summary>
<description>
Extends EL4004 with EtherCAT Working Counter and slave state diagnostics.
When used for I/O, link located fields or their containing buffers to the matching selected PDOs.
The record is not a packed wire buffer; compiler padding is not part of the device specification.
Unlinked/default values do not prove valid I/O. The caller evaluates bus/channel validity before use.
Use one owner task per instance and externally synchronize other access; multi-field snapshots are not atomic.
Copies store data without creating hardware links. Keep borrowed field references valid while consumers are bound.
This passive record performs no validation, synchronization, configuration or protocol advancement.
WcState=TRUE means process-data exchange is invalid. State is acyclic EtherCAT/link information,
not proof of current measurement validity. Link diagnostics to the matching slave InfoData entries.
The selected PDO representation is documented by the base terminal model.
AdsAddr is acyclic mailbox addressing information, not a measurement-validity indicator.
Channels hold raw INT16 output commands; configure electrical range and presentation before use.
</description>
*)
TYPE EL4004_EX EXTENDS EL4004 :
STRUCT
	WcState AT %I* : BOOL;
	State AT %I* : UINT;
	AdsAddr AT %I* : Global.AMSADDR;
END_STRUCT
END_TYPE

// ---- AnalogIO/Outputs/EL4008/EL4008.TcDUT
(*
SPDX-FileCopyrightText: © 2026 Oleksandr Tiutyk <trofimich@gmail.com>
SPDX-License-Identifier: MIT
License: https://opensource.org/license/mit
*)

(*!
<summary>
Beckhoff EL4008: 8-channel analog output terminal (0 .. 10 V, 12-bit).
</summary>
<description>
Process image mapping structure for the EL4008 EtherCAT terminal with 8 analog output channels (0 .. 10 V,
12-bit).
When used for I/O, link located fields or their containing buffers to the matching selected PDOs.
The record is not a packed wire buffer; compiler padding is not part of the device specification.
Unlinked/default values do not prove valid I/O. The caller evaluates bus/channel validity before use.
Use one owner task per instance and externally synchronize other access; multi-field snapshots are not atomic.
Copies store data without creating hardware links. Keep borrowed field references valid while consumers are bound.
This passive record performs no validation, synchronization, configuration or protocol advancement.
Channels hold raw INT16 output commands; configure electrical range and presentation before use.
</description>
*)
TYPE EL4008 :
STRUCT
	Ch1 AT %Q* : INT;
	Ch2 AT %Q* : INT;
	Ch3 AT %Q* : INT;
	Ch4 AT %Q* : INT;
	Ch5 AT %Q* : INT;
	Ch6 AT %Q* : INT;
	Ch7 AT %Q* : INT;
	Ch8 AT %Q* : INT;
END_STRUCT
END_TYPE

// ---- AnalogIO/Outputs/EL4008/EL4008_EX.TcDUT
(*
SPDX-FileCopyrightText: © 2026 Oleksandr Tiutyk <trofimich@gmail.com>
SPDX-License-Identifier: MIT
License: https://opensource.org/license/mit
*)

(*!
<summary>
Beckhoff EL4008_EX: Extended 8-channel analog output terminal with diagnostics.
</summary>
<description>
Extends EL4008 with EtherCAT Working Counter and slave state diagnostics.
When used for I/O, link located fields or their containing buffers to the matching selected PDOs.
The record is not a packed wire buffer; compiler padding is not part of the device specification.
Unlinked/default values do not prove valid I/O. The caller evaluates bus/channel validity before use.
Use one owner task per instance and externally synchronize other access; multi-field snapshots are not atomic.
Copies store data without creating hardware links. Keep borrowed field references valid while consumers are bound.
This passive record performs no validation, synchronization, configuration or protocol advancement.
WcState=TRUE means process-data exchange is invalid. State is acyclic EtherCAT/link information,
not proof of current measurement validity. Link diagnostics to the matching slave InfoData entries.
The selected PDO representation is documented by the base terminal model.
AdsAddr is acyclic mailbox addressing information, not a measurement-validity indicator.
Channels hold raw INT16 output commands; configure electrical range and presentation before use.
</description>
*)
TYPE EL4008_EX EXTENDS EL4008 :
STRUCT
	WcState AT %I* : BOOL;
	State AT %I* : UINT;
	AdsAddr AT %I* : Global.AMSADDR;
END_STRUCT
END_TYPE

// ---- DigitalIO/Inputs/EL1002/EL1002.TcDUT
(*
SPDX-FileCopyrightText: © 2026 Oleksandr Tiutyk <trofimich@gmail.com>
SPDX-License-Identifier: MIT
License: https://opensource.org/license/mit
*)

(*!
<summary>
Beckhoff EL1002: 2-channel digital input terminal (24 V DC, 3 ms filter).
</summary>
<description>
Process image mapping structure for the EL1002 EtherCAT terminal with 2 discrete 24 V DC inputs.
When used for I/O, link located fields or their containing buffers to the matching selected PDOs.
The record is not a packed wire buffer; compiler padding is not part of the device specification.
Unlinked/default values do not prove valid I/O. The caller evaluates bus/channel validity before use.
Use one owner task per instance and externally synchronize other access; multi-field snapshots are not atomic.
Copies store data without creating hardware links. Keep borrowed field references valid while consumers are bound.
This passive record performs no validation, synchronization, configuration or protocol advancement.
</description>
*)
TYPE EL1002 :
STRUCT
	Ch1 AT %I* : BOOL;
	Ch2 AT %I* : BOOL;
END_STRUCT
END_TYPE

// ---- DigitalIO/Inputs/EL1002/EL1002_EX.TcDUT
(*
SPDX-FileCopyrightText: © 2026 Oleksandr Tiutyk <trofimich@gmail.com>
SPDX-License-Identifier: MIT
License: https://opensource.org/license/mit
*)

(*!
<summary>
Beckhoff EL1002_EX: Extended 2-channel digital input terminal with diagnostics.
</summary>
<description>
Extends EL1002 with EtherCAT Working Counter and slave state diagnostics. Note: Simple digital terminals do
not feature CoE mailbox, hence ADS address is not present.
When used for I/O, link located fields or their containing buffers to the matching selected PDOs.
The record is not a packed wire buffer; compiler padding is not part of the device specification.
Unlinked/default values do not prove valid I/O. The caller evaluates bus/channel validity before use.
Use one owner task per instance and externally synchronize other access; multi-field snapshots are not atomic.
Copies store data without creating hardware links. Keep borrowed field references valid while consumers are bound.
This passive record performs no validation, synchronization, configuration or protocol advancement.
WcState=TRUE means process-data exchange is invalid. State is acyclic EtherCAT/link information,
not proof of current measurement validity. Link diagnostics to the matching slave InfoData entries.
The selected PDO representation is documented by the base terminal model.
InputToggle signals an input update by changing state; TRUE alone does not mean fresh data.
</description>
*)
TYPE EL1002_EX EXTENDS EL1002:
STRUCT
	WcState AT %I* : BOOL;
	InputToggle AT %I* : BOOL;
	State AT %I* : UINT;
END_STRUCT
END_TYPE

// ---- DigitalIO/Inputs/EL1004/EL1004.TcDUT
(*
SPDX-FileCopyrightText: © 2026 Oleksandr Tiutyk <trofimich@gmail.com>
SPDX-License-Identifier: MIT
License: https://opensource.org/license/mit
*)

(*!
<summary>
Beckhoff EL1004: 4-channel digital input terminal (24 V DC, 3 ms filter).
</summary>
<description>
Process image mapping structure for the EL1004 EtherCAT terminal with 4 discrete 24 V DC inputs.
When used for I/O, link located fields or their containing buffers to the matching selected PDOs.
The record is not a packed wire buffer; compiler padding is not part of the device specification.
Unlinked/default values do not prove valid I/O. The caller evaluates bus/channel validity before use.
Use one owner task per instance and externally synchronize other access; multi-field snapshots are not atomic.
Copies store data without creating hardware links. Keep borrowed field references valid while consumers are bound.
This passive record performs no validation, synchronization, configuration or protocol advancement.
</description>
*)
TYPE EL1004 :
STRUCT
	Ch1 AT %I* : BOOL;
	Ch2 AT %I* : BOOL;
	Ch3 AT %I* : BOOL;
	Ch4 AT %I* : BOOL;
END_STRUCT
END_TYPE

// ---- DigitalIO/Inputs/EL1004/EL1004_EX.TcDUT
(*
SPDX-FileCopyrightText: © 2026 Oleksandr Tiutyk <trofimich@gmail.com>
SPDX-License-Identifier: MIT
License: https://opensource.org/license/mit
*)

(*!
<summary>
Beckhoff EL1004_EX: Extended 4-channel digital input terminal with diagnostics.
</summary>
<description>
Extends EL1004 with EtherCAT Working Counter and slave state diagnostics.
When used for I/O, link located fields or their containing buffers to the matching selected PDOs.
The record is not a packed wire buffer; compiler padding is not part of the device specification.
Unlinked/default values do not prove valid I/O. The caller evaluates bus/channel validity before use.
Use one owner task per instance and externally synchronize other access; multi-field snapshots are not atomic.
Copies store data without creating hardware links. Keep borrowed field references valid while consumers are bound.
This passive record performs no validation, synchronization, configuration or protocol advancement.
WcState=TRUE means process-data exchange is invalid. State is acyclic EtherCAT/link information,
not proof of current measurement validity. Link diagnostics to the matching slave InfoData entries.
The selected PDO representation is documented by the base terminal model.
InputToggle signals an input update by changing state; TRUE alone does not mean fresh data.
</description>
*)
TYPE EL1004_EX EXTENDS EL1004:
STRUCT
	WcState AT %I* : BOOL;
	InputToggle AT %I* : BOOL;
	State AT %I* : UINT;
END_STRUCT
END_TYPE

// ---- DigitalIO/Inputs/EL1018/EL1018_EX.TcDUT
(*
SPDX-FileCopyrightText: © 2026 Oleksandr Tiutyk <trofimich@gmail.com>
SPDX-License-Identifier: MIT
License: https://opensource.org/license/mit
*)

(*!
<summary>
Beckhoff EL1018_EX: Extended 8-channel fast digital input terminal with diagnostics.
</summary>
<description>
Extends EL1018 with EtherCAT Working Counter and slave state diagnostics.
When used for I/O, link located fields or their containing buffers to the matching selected PDOs.
The record is not a packed wire buffer; compiler padding is not part of the device specification.
Unlinked/default values do not prove valid I/O. The caller evaluates bus/channel validity before use.
Use one owner task per instance and externally synchronize other access; multi-field snapshots are not atomic.
Copies store data without creating hardware links. Keep borrowed field references valid while consumers are bound.
This passive record performs no validation, synchronization, configuration or protocol advancement.
WcState=TRUE means process-data exchange is invalid. State is acyclic EtherCAT/link information,
not proof of current measurement validity. Link diagnostics to the matching slave InfoData entries.
The selected PDO representation is documented by the base terminal model.
InputToggle signals an input update by changing state; TRUE alone does not mean fresh data.
</description>
*)
TYPE EL1018_EX EXTENDS EL1018:
STRUCT
	WcState AT %I* : BOOL;
	InputToggle AT %I* : BOOL;
	State AT %I* : UINT;
END_STRUCT
END_TYPE

// ---- DigitalIO/Inputs/EL1018/EL1018.TcDUT
(*
SPDX-FileCopyrightText: © 2026 Oleksandr Tiutyk <trofimich@gmail.com>
SPDX-License-Identifier: MIT
License: https://opensource.org/license/mit
*)

(*!
<summary>
Beckhoff EL1018: 8-channel fast digital input terminal (24 V DC, 10 µs filter).
</summary>
<description>
Process image mapping structure for the EL1018 fast EtherCAT terminal with 8 discrete 24 V DC inputs and 10
µs input filter.
When used for I/O, link located fields or their containing buffers to the matching selected PDOs.
The record is not a packed wire buffer; compiler padding is not part of the device specification.
Unlinked/default values do not prove valid I/O. The caller evaluates bus/channel validity before use.
Use one owner task per instance and externally synchronize other access; multi-field snapshots are not atomic.
Copies store data without creating hardware links. Keep borrowed field references valid while consumers are bound.
This passive record performs no validation, synchronization, configuration or protocol advancement.
</description>
*)
TYPE EL1018 :
STRUCT
	Ch1 AT %I* : BOOL;
	Ch2 AT %I* : BOOL;
	Ch3 AT %I* : BOOL;
	Ch4 AT %I* : BOOL;
	Ch5 AT %I* : BOOL;
	Ch6 AT %I* : BOOL;
	Ch7 AT %I* : BOOL;
	Ch8 AT %I* : BOOL;
END_STRUCT
END_TYPE

// ---- DigitalIO/Inputs/EL1809/EL1809.TcDUT
(*
SPDX-FileCopyrightText: © 2026 Oleksandr Tiutyk <trofimich@gmail.com>
SPDX-License-Identifier: MIT
License: https://opensource.org/license/mit
*)

(*!
<summary>
Beckhoff EL1809: 16-channel HD digital input terminal (24 V DC, 3 ms filter).
</summary>
<description>
Process image mapping structure for the high-density EL1809 EtherCAT terminal with 16 discrete 24 V DC inputs.
When used for I/O, link located fields or their containing buffers to the matching selected PDOs.
The record is not a packed wire buffer; compiler padding is not part of the device specification.
Unlinked/default values do not prove valid I/O. The caller evaluates bus/channel validity before use.
Use one owner task per instance and externally synchronize other access; multi-field snapshots are not atomic.
Copies store data without creating hardware links. Keep borrowed field references valid while consumers are bound.
This passive record performs no validation, synchronization, configuration or protocol advancement.
</description>
*)
TYPE EL1809 :
STRUCT
	Ch01 AT %I* : BOOL;
	Ch02 AT %I* : BOOL;
	Ch03 AT %I* : BOOL;
	Ch04 AT %I* : BOOL;
	Ch05 AT %I* : BOOL;
	Ch06 AT %I* : BOOL;
	Ch07 AT %I* : BOOL;
	Ch08 AT %I* : BOOL;
	Ch09 AT %I* : BOOL;
	Ch10 AT %I* : BOOL;
	Ch11 AT %I* : BOOL;
	Ch12 AT %I* : BOOL;
	Ch13 AT %I* : BOOL;
	Ch14 AT %I* : BOOL;
	Ch15 AT %I* : BOOL;
	Ch16 AT %I* : BOOL;	
END_STRUCT
END_TYPE

// ---- DigitalIO/Inputs/EL1809/EL1809_EX.TcDUT
(*
SPDX-FileCopyrightText: © 2026 Oleksandr Tiutyk <trofimich@gmail.com>
SPDX-License-Identifier: MIT
License: https://opensource.org/license/mit
*)

(*!
<summary>
Beckhoff EL1809_EX: Extended 16-channel HD digital input terminal with diagnostics.
</summary>
<description>
Extends EL1809 with EtherCAT Working Counter and slave state diagnostics.
When used for I/O, link located fields or their containing buffers to the matching selected PDOs.
The record is not a packed wire buffer; compiler padding is not part of the device specification.
Unlinked/default values do not prove valid I/O. The caller evaluates bus/channel validity before use.
Use one owner task per instance and externally synchronize other access; multi-field snapshots are not atomic.
Copies store data without creating hardware links. Keep borrowed field references valid while consumers are bound.
This passive record performs no validation, synchronization, configuration or protocol advancement.
WcState=TRUE means process-data exchange is invalid. State is acyclic EtherCAT/link information,
not proof of current measurement validity. Link diagnostics to the matching slave InfoData entries.
The selected PDO representation is documented by the base terminal model.
InputToggle signals an input update by changing state; TRUE alone does not mean fresh data.
</description>
*)
TYPE EL1809_EX EXTENDS EL1809:
STRUCT
	WcState AT %I* : BOOL;
	InputToggle AT %I* : BOOL;
	State AT %I* : UINT;
END_STRUCT
END_TYPE

// ---- DigitalIO/Outputs/EL2008/EL2008.TcDUT
(*
SPDX-FileCopyrightText: © 2026 Oleksandr Tiutyk <trofimich@gmail.com>
SPDX-License-Identifier: MIT
License: https://opensource.org/license/mit
*)

(*!
<summary>
Beckhoff EL2008: 8-channel digital output terminal (24 V DC, 0.5 A).
</summary>
<description>
Process image mapping structure for the EL2008 EtherCAT terminal with 8 discrete 24 V DC 0.5 A outputs.
When used for I/O, link located fields or their containing buffers to the matching selected PDOs.
The record is not a packed wire buffer; compiler padding is not part of the device specification.
Unlinked/default values do not prove valid I/O. The caller evaluates bus/channel validity before use.
Use one owner task per instance and externally synchronize other access; multi-field snapshots are not atomic.
Copies store data without creating hardware links. Keep borrowed field references valid while consumers are bound.
This passive record performs no validation, synchronization, configuration or protocol advancement.
</description>
*)
TYPE EL2008 :
STRUCT
	Ch1 AT %Q* : BOOL;
	Ch2 AT %Q* : BOOL;
	Ch3 AT %Q* : BOOL;
	Ch4 AT %Q* : BOOL;
	Ch5 AT %Q* : BOOL;
	Ch6 AT %Q* : BOOL;
	Ch7 AT %Q* : BOOL;
	Ch8 AT %Q* : BOOL;
END_STRUCT
END_TYPE

// ---- DigitalIO/Outputs/EL2008/EL2008_EX.TcDUT
(*
SPDX-FileCopyrightText: © 2026 Oleksandr Tiutyk <trofimich@gmail.com>
SPDX-License-Identifier: MIT
License: https://opensource.org/license/mit
*)

(*!
<summary>
Beckhoff EL2008_EX: Extended 8-channel digital output terminal with diagnostics.
</summary>
<description>
Extends EL2008 with EtherCAT Working Counter and slave state diagnostics.
When used for I/O, link located fields or their containing buffers to the matching selected PDOs.
The record is not a packed wire buffer; compiler padding is not part of the device specification.
Unlinked/default values do not prove valid I/O. The caller evaluates bus/channel validity before use.
Use one owner task per instance and externally synchronize other access; multi-field snapshots are not atomic.
Copies store data without creating hardware links. Keep borrowed field references valid while consumers are bound.
This passive record performs no validation, synchronization, configuration or protocol advancement.
WcState=TRUE means process-data exchange is invalid. State is acyclic EtherCAT/link information,
not proof of current measurement validity. Link diagnostics to the matching slave InfoData entries.
The selected PDO representation is documented by the base terminal model.
</description>
*)
TYPE EL2008_EX EXTENDS EL2008 :
STRUCT
	WcState AT %I* : BOOL;
	State AT %I* : UINT;
END_STRUCT
END_TYPE

// ---- DigitalIO/Outputs/EL2002/EL2002.TcDUT
(*
SPDX-FileCopyrightText: © 2026 Oleksandr Tiutyk <trofimich@gmail.com>
SPDX-License-Identifier: MIT
License: https://opensource.org/license/mit
*)

(*!
<summary>
Beckhoff EL2002: 2-channel digital output terminal (24 V DC, 0.5 A).
</summary>
<description>
Process image mapping structure for the EL2002 EtherCAT terminal with 2 discrete 24 V DC 0.5 A outputs.
When used for I/O, link located fields or their containing buffers to the matching selected PDOs.
The record is not a packed wire buffer; compiler padding is not part of the device specification.
Unlinked/default values do not prove valid I/O. The caller evaluates bus/channel validity before use.
Use one owner task per instance and externally synchronize other access; multi-field snapshots are not atomic.
Copies store data without creating hardware links. Keep borrowed field references valid while consumers are bound.
This passive record performs no validation, synchronization, configuration or protocol advancement.
</description>
*)
TYPE EL2002 :
STRUCT
	Ch1 AT %Q* : BOOL;
	Ch2 AT %Q* : BOOL;
END_STRUCT
END_TYPE

// ---- DigitalIO/Outputs/EL2002/EL2002_EX.TcDUT
(*
SPDX-FileCopyrightText: © 2026 Oleksandr Tiutyk <trofimich@gmail.com>
SPDX-License-Identifier: MIT
License: https://opensource.org/license/mit
*)

(*!
<summary>
Beckhoff EL2002_EX: Extended 2-channel digital output terminal with diagnostics.
</summary>
<description>
Extends EL2002 with EtherCAT Working Counter and slave state diagnostics.
When used for I/O, link located fields or their containing buffers to the matching selected PDOs.
The record is not a packed wire buffer; compiler padding is not part of the device specification.
Unlinked/default values do not prove valid I/O. The caller evaluates bus/channel validity before use.
Use one owner task per instance and externally synchronize other access; multi-field snapshots are not atomic.
Copies store data without creating hardware links. Keep borrowed field references valid while consumers are bound.
This passive record performs no validation, synchronization, configuration or protocol advancement.
WcState=TRUE means process-data exchange is invalid. State is acyclic EtherCAT/link information,
not proof of current measurement validity. Link diagnostics to the matching slave InfoData entries.
The selected PDO representation is documented by the base terminal model.
</description>
*)
TYPE EL2002_EX EXTENDS EL2002 :
STRUCT
	WcState AT %I* : BOOL;
	State AT %I* : UINT;
END_STRUCT
END_TYPE

// ---- DigitalIO/Outputs/EL2004/EL2004.TcDUT
(*
SPDX-FileCopyrightText: © 2026 Oleksandr Tiutyk <trofimich@gmail.com>
SPDX-License-Identifier: MIT
License: https://opensource.org/license/mit
*)

(*!
<summary>
Beckhoff EL2004: 4-channel digital output terminal (24 V DC, 0.5 A).
</summary>
<description>
Process image mapping structure for the EL2004 EtherCAT terminal with 4 discrete 24 V DC 0.5 A outputs.
When used for I/O, link located fields or their containing buffers to the matching selected PDOs.
The record is not a packed wire buffer; compiler padding is not part of the device specification.
Unlinked/default values do not prove valid I/O. The caller evaluates bus/channel validity before use.
Use one owner task per instance and externally synchronize other access; multi-field snapshots are not atomic.
Copies store data without creating hardware links. Keep borrowed field references valid while consumers are bound.
This passive record performs no validation, synchronization, configuration or protocol advancement.
</description>
*)
TYPE EL2004 :
STRUCT
	Ch1 AT %Q* : BOOL;
	Ch2 AT %Q* : BOOL;
	Ch3 AT %Q* : BOOL;
	Ch4 AT %Q* : BOOL;
END_STRUCT
END_TYPE

// ---- DigitalIO/Outputs/EL2004/EL2004_EX.TcDUT
(*
SPDX-FileCopyrightText: © 2026 Oleksandr Tiutyk <trofimich@gmail.com>
SPDX-License-Identifier: MIT
License: https://opensource.org/license/mit
*)

(*!
<summary>
Beckhoff EL2004_EX: Extended 4-channel digital output terminal with diagnostics.
</summary>
<description>
Extends EL2004 with EtherCAT Working Counter and slave state diagnostics.
When used for I/O, link located fields or their containing buffers to the matching selected PDOs.
The record is not a packed wire buffer; compiler padding is not part of the device specification.
Unlinked/default values do not prove valid I/O. The caller evaluates bus/channel validity before use.
Use one owner task per instance and externally synchronize other access; multi-field snapshots are not atomic.
Copies store data without creating hardware links. Keep borrowed field references valid while consumers are bound.
This passive record performs no validation, synchronization, configuration or protocol advancement.
WcState=TRUE means process-data exchange is invalid. State is acyclic EtherCAT/link information,
not proof of current measurement validity. Link diagnostics to the matching slave InfoData entries.
The selected PDO representation is documented by the base terminal model.
</description>
*)
TYPE EL2004_EX EXTENDS EL2004 :
STRUCT
	WcState AT %I* : BOOL;
	State AT %I* : UINT;
END_STRUCT
END_TYPE

// ---- DigitalIO/Outputs/EL2409/EL2409.TcDUT
(*
SPDX-FileCopyrightText: © 2026 Oleksandr Tiutyk <trofimich@gmail.com>
SPDX-License-Identifier: MIT
License: https://opensource.org/license/mit
*)

(*!
<summary>
Beckhoff EL2409: 16-channel HD digital output terminal (24 V DC, 0.5 A, protected).
</summary>
<description>
Process image mapping structure for the high-density EL2409 EtherCAT terminal with 16 discrete 24 V DC 0.5 A
outputs with electronic protection.
When used for I/O, link located fields or their containing buffers to the matching selected PDOs.
The record is not a packed wire buffer; compiler padding is not part of the device specification.
Unlinked/default values do not prove valid I/O. The caller evaluates bus/channel validity before use.
Use one owner task per instance and externally synchronize other access; multi-field snapshots are not atomic.
Copies store data without creating hardware links. Keep borrowed field references valid while consumers are bound.
This passive record performs no validation, synchronization, configuration or protocol advancement.
</description>
*)
TYPE EL2409 :
STRUCT
	Ch01 AT %Q* : BOOL;
	Ch02 AT %Q* : BOOL;
	Ch03 AT %Q* : BOOL;
	Ch04 AT %Q* : BOOL;
	Ch05 AT %Q* : BOOL;
	Ch06 AT %Q* : BOOL;
	Ch07 AT %Q* : BOOL;
	Ch08 AT %Q* : BOOL;
	Ch09 AT %Q* : BOOL;
	Ch10 AT %Q* : BOOL;
	Ch11 AT %Q* : BOOL;
	Ch12 AT %Q* : BOOL;
	Ch13 AT %Q* : BOOL;
	Ch14 AT %Q* : BOOL;
	Ch15 AT %Q* : BOOL;
	Ch16 AT %Q* : BOOL;
END_STRUCT
END_TYPE

// ---- DigitalIO/Outputs/EL2409/EL2409_EX.TcDUT
(*
SPDX-FileCopyrightText: © 2026 Oleksandr Tiutyk <trofimich@gmail.com>
SPDX-License-Identifier: MIT
License: https://opensource.org/license/mit
*)

(*!
<summary>
Beckhoff EL2409_EX: Extended 16-channel HD digital output terminal with diagnostics.
</summary>
<description>
Extends EL2409 with EtherCAT Working Counter and slave state diagnostics.
When used for I/O, link located fields or their containing buffers to the matching selected PDOs.
The record is not a packed wire buffer; compiler padding is not part of the device specification.
Unlinked/default values do not prove valid I/O. The caller evaluates bus/channel validity before use.
Use one owner task per instance and externally synchronize other access; multi-field snapshots are not atomic.
Copies store data without creating hardware links. Keep borrowed field references valid while consumers are bound.
This passive record performs no validation, synchronization, configuration or protocol advancement.
WcState=TRUE means process-data exchange is invalid. State is acyclic EtherCAT/link information,
not proof of current measurement validity. Link diagnostics to the matching slave InfoData entries.
The selected PDO representation is documented by the base terminal model.
</description>
*)
TYPE EL2409_EX EXTENDS EL2409 :
STRUCT
	WcState AT %I* : BOOL;
	State AT %I* : UINT;
END_STRUCT
END_TYPE

// ---- Serial/EL6022/EL6022.TcDUT
(*
SPDX-FileCopyrightText: © 2026 Oleksandr Tiutyk <trofimich@gmail.com>
SPDX-License-Identifier: MIT
License: https://opensource.org/license/mit
*)

(*!
<summary>
Beckhoff EL6022: 2-channel serial interface terminal (RS422 / RS485).
</summary>
<description>
Process image mapping structure for the EL6022 2-channel serial interface terminal using 22-byte data
exchange.
When used for I/O, link located fields or their containing buffers to the matching selected PDOs.
The record is not a packed wire buffer; compiler padding is not part of the device specification.
Unlinked/default values do not prove valid I/O. The caller evaluates bus/channel validity before use.
Use one owner task per instance and externally synchronize other access; multi-field snapshots are not atomic.
Copies store data without creating hardware links. Keep borrowed field references valid while consumers are bound.
This passive record performs no validation, synchronization, configuration or protocol advancement.
Select the 22-byte serial payload with 16-bit status/control words; larger buffers and 9-bit modes
are outside this model. The owning service implements the transmit/receive toggle handshake.
</description>
*)
TYPE EL6022 :
STRUCT
	Ch1 : EL6022_CHANNEL;
	Ch2 : EL6022_CHANNEL;
END_STRUCT
END_TYPE

// ---- Serial/EL6022/EL6022_CHANNEL.TcDUT
(*
SPDX-FileCopyrightText: © 2026 Oleksandr Tiutyk <trofimich@gmail.com>
SPDX-License-Identifier: MIT
License: https://opensource.org/license/mit
*)

(*!
<summary>
Beckhoff EL6022: Serial communication channel process image.
</summary>
<description>
Encapsulates 22-byte input (InData) and output (OutData) process data for one RS422/RS485 communication
channel.
When used for I/O, link located fields or their containing buffers to the matching selected PDOs.
The record is not a packed wire buffer; compiler padding is not part of the device specification.
Unlinked/default values do not prove valid I/O. The caller evaluates bus/channel validity before use.
Use one owner task per instance and externally synchronize other access; multi-field snapshots are not atomic.
Copies store data without creating hardware links. Keep borrowed field references valid while consumers are bound.
This passive record performs no validation, synchronization, configuration or protocol advancement.
Select the 22-byte serial payload with 16-bit status/control words; larger buffers and 9-bit modes
are outside this model. The owning service implements the transmit/receive toggle handshake.
</description>
*)
TYPE EL6022_CHANNEL :
STRUCT
	InData AT %I* : EL6xxx22ByteInData;
	OutData AT %Q* : EL6xxx22ByteOutData;
END_STRUCT
END_TYPE

// ---- Serial/EL6022/EL6022_EX.TcDUT
(*
SPDX-FileCopyrightText: © 2026 Oleksandr Tiutyk <trofimich@gmail.com>
SPDX-License-Identifier: MIT
License: https://opensource.org/license/mit
*)

(*!
<summary>
Beckhoff EL6022_EX: Extended 2-channel serial interface terminal with diagnostics.
</summary>
<description>
Extends EL6022 with EtherCAT Working Counter, slave state, and CoE mailbox ADS address diagnostics.
When used for I/O, link located fields or their containing buffers to the matching selected PDOs.
The record is not a packed wire buffer; compiler padding is not part of the device specification.
Unlinked/default values do not prove valid I/O. The caller evaluates bus/channel validity before use.
Use one owner task per instance and externally synchronize other access; multi-field snapshots are not atomic.
Copies store data without creating hardware links. Keep borrowed field references valid while consumers are bound.
This passive record performs no validation, synchronization, configuration or protocol advancement.
WcState=TRUE means process-data exchange is invalid. State is acyclic EtherCAT/link information,
not proof of current measurement validity. Link diagnostics to the matching slave InfoData entries.
The selected PDO representation is documented by the base terminal model.
InputToggle signals an input update by changing state; TRUE alone does not mean fresh data.
AdsAddr is acyclic mailbox addressing information, not a measurement-validity indicator.
Select the 22-byte serial payload with 16-bit status/control words; larger buffers and 9-bit modes
are outside this model. The owning service implements the transmit/receive toggle handshake.
</description>
*)
TYPE EL6022_EX EXTENDS EL6022 :
STRUCT
	WcState AT %I* : BOOL;
	InputToggle AT %I* : BOOL;
	State AT %I* : UINT;
	AdsAddr AT %I* : Global.AMSADDR;
END_STRUCT
END_TYPE

// ---- Serial/EL6xxx22ByteInData.TcDUT
(*
SPDX-FileCopyrightText: © 2026 Oleksandr Tiutyk <trofimich@gmail.com>
SPDX-License-Identifier: MIT
License: https://opensource.org/license/mit
*)

(*!
<summary>
Beckhoff EL6xxx: 22-byte serial communication input process image.
</summary>
<description>
Encapsulates a 16-bit status word and a 22-byte received data buffer for EL6xxx serial interface terminals.
When used for I/O, link located fields or their containing buffers to the matching selected PDOs.
The record is not a packed wire buffer; compiler padding is not part of the device specification.
Unlinked/default values do not prove valid I/O. The caller evaluates bus/channel validity before use.
Use one owner task per instance and externally synchronize other access; multi-field snapshots are not atomic.
Copies store data without creating hardware links. Keep borrowed field references valid while consumers are bound.
This passive record performs no validation, synchronization, configuration or protocol advancement.
Select the 22-byte serial payload with 16-bit status/control words; larger buffers and 9-bit modes
are outside this model. The owning service implements the transmit/receive toggle handshake.
</description>
*)
TYPE EL6xxx22ByteInData :
STRUCT
	Status : WORD;     
	Data : ARRAY [0..21] OF BYTE; 
END_STRUCT
END_TYPE

// ---- Serial/EL6xxx22ByteOutData.TcDUT
(*
SPDX-FileCopyrightText: © 2026 Oleksandr Tiutyk <trofimich@gmail.com>
SPDX-License-Identifier: MIT
License: https://opensource.org/license/mit
*)

(*!
<summary>
Beckhoff EL6xxx: 22-byte serial communication output process image.
</summary>
<description>
Encapsulates a 16-bit control word and a 22-byte transmit data buffer for EL6xxx serial interface terminals.
When used for I/O, link located fields or their containing buffers to the matching selected PDOs.
The record is not a packed wire buffer; compiler padding is not part of the device specification.
Unlinked/default values do not prove valid I/O. The caller evaluates bus/channel validity before use.
Use one owner task per instance and externally synchronize other access; multi-field snapshots are not atomic.
Copies store data without creating hardware links. Keep borrowed field references valid while consumers are bound.
This passive record performs no validation, synchronization, configuration or protocol advancement.
Select the 22-byte serial payload with 16-bit status/control words; larger buffers and 9-bit modes
are outside this model. The owning service implements the transmit/receive toggle handshake.
</description>
*)
TYPE EL6xxx22ByteOutData :
STRUCT
	Control : WORD;     
	Data : ARRAY [0..21] OF BYTE; 
END_STRUCT
END_TYPE

// ---- AnalogIO/Inputs/RTD_INPUT_CHANNEL.TcDUT
(*
SPDX-FileCopyrightText: © 2026 Oleksandr Tiutyk <trofimich@gmail.com>
SPDX-License-Identifier: MIT
License: https://opensource.org/license/mit
*)

(*!
<summary>
Beckhoff RTD temperature sensor channel process image.
</summary>
<description>
Represents the standard 16-bit status plus INT16 measured-value PDO, not the compact value-only PDO.
Default temperature presentation is 0.1 deg C per digit; high resolution is 0.01 deg C per digit.
Thus raw 253 means 25.3 or 2.53 deg C respectively. Configure presentation explicitly.
Signed-amount or resistance presentations require their matching interpretation; this type stores raw bits.
Check channel status before using Value. This record does not choose or convert device presentation.
When used for I/O, link located fields or their containing buffers to the matching selected PDOs.
The record is not a packed wire buffer; compiler padding is not part of the device specification.
Unlinked/default values do not prove valid I/O. The caller evaluates bus/channel validity before use.
Use one owner task per instance and externally synchronize other access; multi-field snapshots are not atomic.
Copies store data without creating hardware links. Keep borrowed field references valid while consumers are bound.
This passive record performs no validation, synchronization, configuration or protocol advancement.
</description>
*)
TYPE RTD_INPUT_CHANNEL :
STRUCT
	Status AT %I* : WORD;
	Value AT %I* : INT;
END_STRUCT
END_TYPE

// ---- AnalogIO/Inputs/THERMOCOUPLE_INPUT_CHANNEL.TcDUT
(*
SPDX-FileCopyrightText: © 2026 Oleksandr Tiutyk <trofimich@gmail.com>
SPDX-License-Identifier: MIT
License: https://opensource.org/license/mit
*)

(*!
<summary>
Beckhoff Thermocouple temperature sensor channel process image.
</summary>
<description>
Represents the standard 16-bit status plus INT16 temperature PDO, not the compact value-only PDO.
Default presentation is 0.1 deg C per digit; high resolution is 0.01 deg C per digit.
Thus raw 253 means 25.3 or 2.53 deg C respectively. Configure presentation explicitly.
Signed-amount presentation requires its matching interpretation; this type stores raw bits.
Check channel status before using Value. Cold-junction compensation follows device configuration.
When used for I/O, link located fields or their containing buffers to the matching selected PDOs.
The record is not a packed wire buffer; compiler padding is not part of the device specification.
Unlinked/default values do not prove valid I/O. The caller evaluates bus/channel validity before use.
Use one owner task per instance and externally synchronize other access; multi-field snapshots are not atomic.
Copies store data without creating hardware links. Keep borrowed field references valid while consumers are bound.
This passive record performs no validation, synchronization, configuration or protocol advancement.
</description>
*)
TYPE THERMOCOUPLE_INPUT_CHANNEL :
STRUCT
	Status AT %I* : WORD;
	Value AT %I* : INT;
END_STRUCT
END_TYPE

// ---- AnalogIO/Inputs/EL3201/EL3201.TcDUT
(*
SPDX-FileCopyrightText: © 2026 Oleksandr Tiutyk <trofimich@gmail.com>
SPDX-License-Identifier: MIT
License: https://opensource.org/license/mit
*)

(*!
<summary>
Beckhoff EL3201: 1-channel RTD resistance thermometer terminal (Pt100, Pt1000, Ni120...).
</summary>
<description>
Process image mapping structure for the EL3201 1-channel RTD temperature input terminal.
When used for I/O, link located fields or their containing buffers to the matching selected PDOs.
The record is not a packed wire buffer; compiler padding is not part of the device specification.
Unlinked/default values do not prove valid I/O. The caller evaluates bus/channel validity before use.
Use one owner task per instance and externally synchronize other access; multi-field snapshots are not atomic.
Copies store data without creating hardware links. Keep borrowed field references valid while consumers are bound.
This passive record performs no validation, synchronization, configuration or protocol advancement.
Select standard status-plus-INT16 PDOs; compact layouts are unsupported. Configure presentation explicitly:
0.1/0.01 deg C per digit follows the device setting, not this record.
</description>
*)
TYPE EL3201 :
STRUCT
	Ch1 : RTD_INPUT_CHANNEL;
END_STRUCT
END_TYPE

// ---- AnalogIO/Inputs/EL3201/EL3201_EX.TcDUT
(*
SPDX-FileCopyrightText: © 2026 Oleksandr Tiutyk <trofimich@gmail.com>
SPDX-License-Identifier: MIT
License: https://opensource.org/license/mit
*)

(*!
<summary>
Beckhoff EL3201_EX: Extended 1-channel RTD terminal with diagnostics.
</summary>
<description>
Extends EL3201 with EtherCAT Working Counter, slave state, and CoE mailbox ADS address diagnostics.
When used for I/O, link located fields or their containing buffers to the matching selected PDOs.
The record is not a packed wire buffer; compiler padding is not part of the device specification.
Unlinked/default values do not prove valid I/O. The caller evaluates bus/channel validity before use.
Use one owner task per instance and externally synchronize other access; multi-field snapshots are not atomic.
Copies store data without creating hardware links. Keep borrowed field references valid while consumers are bound.
This passive record performs no validation, synchronization, configuration or protocol advancement.
WcState=TRUE means process-data exchange is invalid. State is acyclic EtherCAT/link information,
not proof of current measurement validity. Link diagnostics to the matching slave InfoData entries.
The selected PDO representation is documented by the base terminal model.
InputToggle signals an input update by changing state; TRUE alone does not mean fresh data.
AdsAddr is acyclic mailbox addressing information, not a measurement-validity indicator.
Select standard status-plus-INT16 PDOs; compact layouts are unsupported. Configure presentation explicitly:
0.1/0.01 deg C per digit follows the device setting, not this record.
</description>
*)
TYPE EL3201_EX EXTENDS EL3201 :
STRUCT
	WcState AT %I* : BOOL;
	InputToggle AT %I* : BOOL;
	State AT %I* : UINT;
	AdsAddr AT %I* : Global.AMSADDR;
END_STRUCT
END_TYPE

// ---- AnalogIO/Inputs/EL3202/EL3202.TcDUT
(*
SPDX-FileCopyrightText: © 2026 Oleksandr Tiutyk <trofimich@gmail.com>
SPDX-License-Identifier: MIT
License: https://opensource.org/license/mit
*)

(*!
<summary>
Beckhoff EL3202: 2-channel RTD resistance thermometer terminal (Pt100, Pt1000, Ni120...).
</summary>
<description>
Process image mapping structure for the EL3202 2-channel RTD temperature input terminal.
When used for I/O, link located fields or their containing buffers to the matching selected PDOs.
The record is not a packed wire buffer; compiler padding is not part of the device specification.
Unlinked/default values do not prove valid I/O. The caller evaluates bus/channel validity before use.
Use one owner task per instance and externally synchronize other access; multi-field snapshots are not atomic.
Copies store data without creating hardware links. Keep borrowed field references valid while consumers are bound.
This passive record performs no validation, synchronization, configuration or protocol advancement.
Select standard status-plus-INT16 PDOs; compact layouts are unsupported. Configure presentation explicitly:
0.1/0.01 deg C per digit follows the device setting, not this record.
</description>
*)
TYPE EL3202 :
STRUCT
	Ch1 : RTD_INPUT_CHANNEL;
	Ch2 : RTD_INPUT_CHANNEL;
END_STRUCT
END_TYPE

// ---- AnalogIO/Inputs/EL3202/EL3202_EX.TcDUT
(*
SPDX-FileCopyrightText: © 2026 Oleksandr Tiutyk <trofimich@gmail.com>
SPDX-License-Identifier: MIT
License: https://opensource.org/license/mit
*)

(*!
<summary>
Beckhoff EL3202_EX: Extended 2-channel RTD terminal with diagnostics.
</summary>
<description>
Extends EL3202 with EtherCAT Working Counter, slave state, and CoE mailbox ADS address diagnostics.
When used for I/O, link located fields or their containing buffers to the matching selected PDOs.
The record is not a packed wire buffer; compiler padding is not part of the device specification.
Unlinked/default values do not prove valid I/O. The caller evaluates bus/channel validity before use.
Use one owner task per instance and externally synchronize other access; multi-field snapshots are not atomic.
Copies store data without creating hardware links. Keep borrowed field references valid while consumers are bound.
This passive record performs no validation, synchronization, configuration or protocol advancement.
WcState=TRUE means process-data exchange is invalid. State is acyclic EtherCAT/link information,
not proof of current measurement validity. Link diagnostics to the matching slave InfoData entries.
The selected PDO representation is documented by the base terminal model.
InputToggle signals an input update by changing state; TRUE alone does not mean fresh data.
AdsAddr is acyclic mailbox addressing information, not a measurement-validity indicator.
Select standard status-plus-INT16 PDOs; compact layouts are unsupported. Configure presentation explicitly:
0.1/0.01 deg C per digit follows the device setting, not this record.
</description>
*)
TYPE EL3202_EX EXTENDS EL3202 :
STRUCT
	WcState AT %I* : BOOL;
	InputToggle AT %I* : BOOL;
	State AT %I* : UINT;
	AdsAddr AT %I* : Global.AMSADDR;
END_STRUCT
END_TYPE

// ---- AnalogIO/Inputs/EL3204/EL3204.TcDUT
(*
SPDX-FileCopyrightText: © 2026 Oleksandr Tiutyk <trofimich@gmail.com>
SPDX-License-Identifier: MIT
License: https://opensource.org/license/mit
*)

(*!
<summary>
Beckhoff EL3204: 4-channel RTD resistance thermometer terminal (Pt100, Pt1000, Ni120...).
</summary>
<description>
Process image mapping structure for the EL3204 4-channel RTD temperature input terminal.
When used for I/O, link located fields or their containing buffers to the matching selected PDOs.
The record is not a packed wire buffer; compiler padding is not part of the device specification.
Unlinked/default values do not prove valid I/O. The caller evaluates bus/channel validity before use.
Use one owner task per instance and externally synchronize other access; multi-field snapshots are not atomic.
Copies store data without creating hardware links. Keep borrowed field references valid while consumers are bound.
This passive record performs no validation, synchronization, configuration or protocol advancement.
Select standard status-plus-INT16 PDOs; compact layouts are unsupported. Configure presentation explicitly:
0.1/0.01 deg C per digit follows the device setting, not this record.
</description>
*)
TYPE EL3204 :
STRUCT
	Ch1 : RTD_INPUT_CHANNEL;
	Ch2 : RTD_INPUT_CHANNEL;
	Ch3 : RTD_INPUT_CHANNEL;
	Ch4 : RTD_INPUT_CHANNEL;
END_STRUCT
END_TYPE

// ---- AnalogIO/Inputs/EL3204/EL3204_EX.TcDUT
(*
SPDX-FileCopyrightText: © 2026 Oleksandr Tiutyk <trofimich@gmail.com>
SPDX-License-Identifier: MIT
License: https://opensource.org/license/mit
*)

(*!
<summary>
Beckhoff EL3204_EX: Extended 4-channel RTD terminal with diagnostics.
</summary>
<description>
Extends EL3204 with EtherCAT Working Counter, slave state, and CoE mailbox ADS address diagnostics.
When used for I/O, link located fields or their containing buffers to the matching selected PDOs.
The record is not a packed wire buffer; compiler padding is not part of the device specification.
Unlinked/default values do not prove valid I/O. The caller evaluates bus/channel validity before use.
Use one owner task per instance and externally synchronize other access; multi-field snapshots are not atomic.
Copies store data without creating hardware links. Keep borrowed field references valid while consumers are bound.
This passive record performs no validation, synchronization, configuration or protocol advancement.
WcState=TRUE means process-data exchange is invalid. State is acyclic EtherCAT/link information,
not proof of current measurement validity. Link diagnostics to the matching slave InfoData entries.
The selected PDO representation is documented by the base terminal model.
InputToggle signals an input update by changing state; TRUE alone does not mean fresh data.
AdsAddr is acyclic mailbox addressing information, not a measurement-validity indicator.
Select standard status-plus-INT16 PDOs; compact layouts are unsupported. Configure presentation explicitly:
0.1/0.01 deg C per digit follows the device setting, not this record.
</description>
*)
TYPE EL3204_EX EXTENDS EL3204 :
STRUCT
	WcState AT %I* : BOOL;
	InputToggle AT %I* : BOOL;
	State AT %I* : UINT;
	AdsAddr AT %I* : Global.AMSADDR;
END_STRUCT
END_TYPE

// ---- AnalogIO/Inputs/EL3208/EL3208.TcDUT
(*
SPDX-FileCopyrightText: © 2026 Oleksandr Tiutyk <trofimich@gmail.com>
SPDX-License-Identifier: MIT
License: https://opensource.org/license/mit
*)

(*!
<summary>
Beckhoff EL3208: 8-channel RTD resistance thermometer terminal (Pt100, Pt1000, Ni120...).
</summary>
<description>
Process image mapping structure for the EL3208 8-channel RTD temperature input terminal.
When used for I/O, link located fields or their containing buffers to the matching selected PDOs.
The record is not a packed wire buffer; compiler padding is not part of the device specification.
Unlinked/default values do not prove valid I/O. The caller evaluates bus/channel validity before use.
Use one owner task per instance and externally synchronize other access; multi-field snapshots are not atomic.
Copies store data without creating hardware links. Keep borrowed field references valid while consumers are bound.
This passive record performs no validation, synchronization, configuration or protocol advancement.
Select standard status-plus-INT16 PDOs; compact layouts are unsupported. Configure presentation explicitly:
0.1/0.01 deg C per digit follows the device setting, not this record.
</description>
*)
TYPE EL3208 :
STRUCT
	Ch1 : RTD_INPUT_CHANNEL;
	Ch2 : RTD_INPUT_CHANNEL;
	Ch3 : RTD_INPUT_CHANNEL;
	Ch4 : RTD_INPUT_CHANNEL;
	Ch5 : RTD_INPUT_CHANNEL;
	Ch6 : RTD_INPUT_CHANNEL;
	Ch7 : RTD_INPUT_CHANNEL;
	Ch8 : RTD_INPUT_CHANNEL;
END_STRUCT
END_TYPE

// ---- AnalogIO/Inputs/EL3208/EL3208_EX.TcDUT
(*
SPDX-FileCopyrightText: © 2026 Oleksandr Tiutyk <trofimich@gmail.com>
SPDX-License-Identifier: MIT
License: https://opensource.org/license/mit
*)

(*!
<summary>
Beckhoff EL3208_EX: Extended 8-channel RTD terminal with diagnostics.
</summary>
<description>
Extends EL3208 with EtherCAT Working Counter, slave state, and CoE mailbox ADS address diagnostics.
When used for I/O, link located fields or their containing buffers to the matching selected PDOs.
The record is not a packed wire buffer; compiler padding is not part of the device specification.
Unlinked/default values do not prove valid I/O. The caller evaluates bus/channel validity before use.
Use one owner task per instance and externally synchronize other access; multi-field snapshots are not atomic.
Copies store data without creating hardware links. Keep borrowed field references valid while consumers are bound.
This passive record performs no validation, synchronization, configuration or protocol advancement.
WcState=TRUE means process-data exchange is invalid. State is acyclic EtherCAT/link information,
not proof of current measurement validity. Link diagnostics to the matching slave InfoData entries.
The selected PDO representation is documented by the base terminal model.
InputToggle signals an input update by changing state; TRUE alone does not mean fresh data.
AdsAddr is acyclic mailbox addressing information, not a measurement-validity indicator.
Select standard status-plus-INT16 PDOs; compact layouts are unsupported. Configure presentation explicitly:
0.1/0.01 deg C per digit follows the device setting, not this record.
</description>
*)
TYPE EL3208_EX EXTENDS EL3208 :
STRUCT
	WcState AT %I* : BOOL;
	InputToggle AT %I* : BOOL;
	State AT %I* : UINT;
	AdsAddr AT %I* : Global.AMSADDR;
END_STRUCT
END_TYPE

// ---- AnalogIO/Inputs/EL3311/EL3311.TcDUT
(*
SPDX-FileCopyrightText: © 2026 Oleksandr Tiutyk <trofimich@gmail.com>
SPDX-License-Identifier: MIT
License: https://opensource.org/license/mit
*)

(*!
<summary>
Beckhoff EL3311: 1-channel thermocouple input terminal (J, K, T, E, N, R, S, B, C).
</summary>
<description>
Process image mapping structure for the EL3311 1-channel thermocouple input terminal.
When used for I/O, link located fields or their containing buffers to the matching selected PDOs.
The record is not a packed wire buffer; compiler padding is not part of the device specification.
Unlinked/default values do not prove valid I/O. The caller evaluates bus/channel validity before use.
Use one owner task per instance and externally synchronize other access; multi-field snapshots are not atomic.
Copies store data without creating hardware links. Keep borrowed field references valid while consumers are bound.
This passive record performs no validation, synchronization, configuration or protocol advancement.
Select standard status-plus-INT16 PDOs; compact layouts are unsupported. Configure presentation explicitly:
0.1/0.01 deg C per digit follows the device setting, not this record.
</description>
*)
TYPE EL3311 :
STRUCT
	Ch1 : THERMOCOUPLE_INPUT_CHANNEL;
END_STRUCT
END_TYPE

// ---- AnalogIO/Inputs/EL3311/EL3311_EX.TcDUT
(*
SPDX-FileCopyrightText: © 2026 Oleksandr Tiutyk <trofimich@gmail.com>
SPDX-License-Identifier: MIT
License: https://opensource.org/license/mit
*)

(*!
<summary>
Beckhoff EL3311_EX: Extended 1-channel thermocouple terminal with diagnostics.
</summary>
<description>
Extends EL3311 with EtherCAT Working Counter, slave state, and CoE mailbox ADS address diagnostics.
When used for I/O, link located fields or their containing buffers to the matching selected PDOs.
The record is not a packed wire buffer; compiler padding is not part of the device specification.
Unlinked/default values do not prove valid I/O. The caller evaluates bus/channel validity before use.
Use one owner task per instance and externally synchronize other access; multi-field snapshots are not atomic.
Copies store data without creating hardware links. Keep borrowed field references valid while consumers are bound.
This passive record performs no validation, synchronization, configuration or protocol advancement.
WcState=TRUE means process-data exchange is invalid. State is acyclic EtherCAT/link information,
not proof of current measurement validity. Link diagnostics to the matching slave InfoData entries.
The selected PDO representation is documented by the base terminal model.
InputToggle signals an input update by changing state; TRUE alone does not mean fresh data.
AdsAddr is acyclic mailbox addressing information, not a measurement-validity indicator.
Select standard status-plus-INT16 PDOs; compact layouts are unsupported. Configure presentation explicitly:
0.1/0.01 deg C per digit follows the device setting, not this record.
</description>
*)
TYPE EL3311_EX EXTENDS EL3311 :
STRUCT
	WcState AT %I* : BOOL;
	InputToggle AT %I* : BOOL;
	State AT %I* : UINT;
	AdsAddr AT %I* : Global.AMSADDR;
END_STRUCT
END_TYPE

// ---- AnalogIO/Inputs/EL3312/EL3312.TcDUT
(*
SPDX-FileCopyrightText: © 2026 Oleksandr Tiutyk <trofimich@gmail.com>
SPDX-License-Identifier: MIT
License: https://opensource.org/license/mit
*)

(*!
<summary>
Beckhoff EL3312: 2-channel thermocouple input terminal (J, K, T, E, N, R, S, B, C).
</summary>
<description>
Process image mapping structure for the EL3312 2-channel thermocouple input terminal.
When used for I/O, link located fields or their containing buffers to the matching selected PDOs.
The record is not a packed wire buffer; compiler padding is not part of the device specification.
Unlinked/default values do not prove valid I/O. The caller evaluates bus/channel validity before use.
Use one owner task per instance and externally synchronize other access; multi-field snapshots are not atomic.
Copies store data without creating hardware links. Keep borrowed field references valid while consumers are bound.
This passive record performs no validation, synchronization, configuration or protocol advancement.
Select standard status-plus-INT16 PDOs; compact layouts are unsupported. Configure presentation explicitly:
0.1/0.01 deg C per digit follows the device setting, not this record.
</description>
*)
TYPE EL3312 :
STRUCT
	Ch1 : THERMOCOUPLE_INPUT_CHANNEL;
	Ch2 : THERMOCOUPLE_INPUT_CHANNEL;
END_STRUCT
END_TYPE

// ---- AnalogIO/Inputs/EL3312/EL3312_EX.TcDUT
(*
SPDX-FileCopyrightText: © 2026 Oleksandr Tiutyk <trofimich@gmail.com>
SPDX-License-Identifier: MIT
License: https://opensource.org/license/mit
*)

(*!
<summary>
Beckhoff EL3312_EX: Extended 2-channel thermocouple terminal with diagnostics.
</summary>
<description>
Extends EL3312 with EtherCAT Working Counter, slave state, and CoE mailbox ADS address diagnostics.
When used for I/O, link located fields or their containing buffers to the matching selected PDOs.
The record is not a packed wire buffer; compiler padding is not part of the device specification.
Unlinked/default values do not prove valid I/O. The caller evaluates bus/channel validity before use.
Use one owner task per instance and externally synchronize other access; multi-field snapshots are not atomic.
Copies store data without creating hardware links. Keep borrowed field references valid while consumers are bound.
This passive record performs no validation, synchronization, configuration or protocol advancement.
WcState=TRUE means process-data exchange is invalid. State is acyclic EtherCAT/link information,
not proof of current measurement validity. Link diagnostics to the matching slave InfoData entries.
The selected PDO representation is documented by the base terminal model.
InputToggle signals an input update by changing state; TRUE alone does not mean fresh data.
AdsAddr is acyclic mailbox addressing information, not a measurement-validity indicator.
Select standard status-plus-INT16 PDOs; compact layouts are unsupported. Configure presentation explicitly:
0.1/0.01 deg C per digit follows the device setting, not this record.
</description>
*)
TYPE EL3312_EX EXTENDS EL3312 :
STRUCT
	WcState AT %I* : BOOL;
	InputToggle AT %I* : BOOL;
	State AT %I* : UINT;
	AdsAddr AT %I* : Global.AMSADDR;
END_STRUCT
END_TYPE

// ---- AnalogIO/Inputs/EL3314/EL3314.TcDUT
(*
SPDX-FileCopyrightText: © 2026 Oleksandr Tiutyk <trofimich@gmail.com>
SPDX-License-Identifier: MIT
License: https://opensource.org/license/mit
*)

(*!
<summary>
Beckhoff EL3314: 4-channel thermocouple input terminal (J, K, T, E, N, R, S, B, C).
</summary>
<description>
Process image mapping structure for the EL3314 4-channel thermocouple input terminal.
When used for I/O, link located fields or their containing buffers to the matching selected PDOs.
The record is not a packed wire buffer; compiler padding is not part of the device specification.
Unlinked/default values do not prove valid I/O. The caller evaluates bus/channel validity before use.
Use one owner task per instance and externally synchronize other access; multi-field snapshots are not atomic.
Copies store data without creating hardware links. Keep borrowed field references valid while consumers are bound.
This passive record performs no validation, synchronization, configuration or protocol advancement.
Select standard status-plus-INT16 PDOs; compact layouts are unsupported. Configure presentation explicitly:
0.1/0.01 deg C per digit follows the device setting, not this record.
</description>
*)
TYPE EL3314 :
STRUCT
	Ch1 : THERMOCOUPLE_INPUT_CHANNEL;
	Ch2 : THERMOCOUPLE_INPUT_CHANNEL;
	Ch3 : THERMOCOUPLE_INPUT_CHANNEL;
	Ch4 : THERMOCOUPLE_INPUT_CHANNEL;
END_STRUCT
END_TYPE

// ---- AnalogIO/Inputs/EL3314/EL3314_EX.TcDUT
(*
SPDX-FileCopyrightText: © 2026 Oleksandr Tiutyk <trofimich@gmail.com>
SPDX-License-Identifier: MIT
License: https://opensource.org/license/mit
*)

(*!
<summary>
Beckhoff EL3314_EX: Extended 4-channel thermocouple terminal with diagnostics.
</summary>
<description>
Extends EL3314 with EtherCAT Working Counter, slave state, and CoE mailbox ADS address diagnostics.
When used for I/O, link located fields or their containing buffers to the matching selected PDOs.
The record is not a packed wire buffer; compiler padding is not part of the device specification.
Unlinked/default values do not prove valid I/O. The caller evaluates bus/channel validity before use.
Use one owner task per instance and externally synchronize other access; multi-field snapshots are not atomic.
Copies store data without creating hardware links. Keep borrowed field references valid while consumers are bound.
This passive record performs no validation, synchronization, configuration or protocol advancement.
WcState=TRUE means process-data exchange is invalid. State is acyclic EtherCAT/link information,
not proof of current measurement validity. Link diagnostics to the matching slave InfoData entries.
The selected PDO representation is documented by the base terminal model.
InputToggle signals an input update by changing state; TRUE alone does not mean fresh data.
AdsAddr is acyclic mailbox addressing information, not a measurement-validity indicator.
Select standard status-plus-INT16 PDOs; compact layouts are unsupported. Configure presentation explicitly:
0.1/0.01 deg C per digit follows the device setting, not this record.
</description>
*)
TYPE EL3314_EX EXTENDS EL3314 :
STRUCT
	WcState AT %I* : BOOL;
	InputToggle AT %I* : BOOL;
	State AT %I* : UINT;
	AdsAddr AT %I* : Global.AMSADDR;
END_STRUCT
END_TYPE

// ---- AnalogIO/Inputs/EL3318/EL3318.TcDUT
(*
SPDX-FileCopyrightText: © 2026 Oleksandr Tiutyk <trofimich@gmail.com>
SPDX-License-Identifier: MIT
License: https://opensource.org/license/mit
*)

(*!
<summary>
Beckhoff EL3318: 8-channel thermocouple input terminal (J, K, T, E, N, R, S, B, C).
</summary>
<description>
Process image mapping structure for the EL3318 8-channel thermocouple input terminal.
When used for I/O, link located fields or their containing buffers to the matching selected PDOs.
The record is not a packed wire buffer; compiler padding is not part of the device specification.
Unlinked/default values do not prove valid I/O. The caller evaluates bus/channel validity before use.
Use one owner task per instance and externally synchronize other access; multi-field snapshots are not atomic.
Copies store data without creating hardware links. Keep borrowed field references valid while consumers are bound.
This passive record performs no validation, synchronization, configuration or protocol advancement.
Select standard status-plus-INT16 PDOs; compact layouts are unsupported. Configure presentation explicitly:
0.1/0.01 deg C per digit follows the device setting, not this record.
</description>
*)
TYPE EL3318 :
STRUCT
	Ch1 : THERMOCOUPLE_INPUT_CHANNEL;
	Ch2 : THERMOCOUPLE_INPUT_CHANNEL;
	Ch3 : THERMOCOUPLE_INPUT_CHANNEL;
	Ch4 : THERMOCOUPLE_INPUT_CHANNEL;
	Ch5 : THERMOCOUPLE_INPUT_CHANNEL;
	Ch6 : THERMOCOUPLE_INPUT_CHANNEL;
	Ch7 : THERMOCOUPLE_INPUT_CHANNEL;
	Ch8 : THERMOCOUPLE_INPUT_CHANNEL;
END_STRUCT
END_TYPE

// ---- AnalogIO/Inputs/EL3318/EL3318_EX.TcDUT
(*
SPDX-FileCopyrightText: © 2026 Oleksandr Tiutyk <trofimich@gmail.com>
SPDX-License-Identifier: MIT
License: https://opensource.org/license/mit
*)

(*!
<summary>
Beckhoff EL3318_EX: Extended 8-channel thermocouple terminal with diagnostics.
</summary>
<description>
Extends EL3318 with EtherCAT Working Counter, slave state, and CoE mailbox ADS address diagnostics.
When used for I/O, link located fields or their containing buffers to the matching selected PDOs.
The record is not a packed wire buffer; compiler padding is not part of the device specification.
Unlinked/default values do not prove valid I/O. The caller evaluates bus/channel validity before use.
Use one owner task per instance and externally synchronize other access; multi-field snapshots are not atomic.
Copies store data without creating hardware links. Keep borrowed field references valid while consumers are bound.
This passive record performs no validation, synchronization, configuration or protocol advancement.
WcState=TRUE means process-data exchange is invalid. State is acyclic EtherCAT/link information,
not proof of current measurement validity. Link diagnostics to the matching slave InfoData entries.
The selected PDO representation is documented by the base terminal model.
InputToggle signals an input update by changing state; TRUE alone does not mean fresh data.
AdsAddr is acyclic mailbox addressing information, not a measurement-validity indicator.
Select standard status-plus-INT16 PDOs; compact layouts are unsupported. Configure presentation explicitly:
0.1/0.01 deg C per digit follows the device setting, not this record.
</description>
*)
TYPE EL3318_EX EXTENDS EL3318 :
STRUCT
	WcState AT %I* : BOOL;
	InputToggle AT %I* : BOOL;
	State AT %I* : UINT;
	AdsAddr AT %I* : Global.AMSADDR;
END_STRUCT
END_TYPE

// ---- DigitalIO/Inputs/EL1008/EL1008.TcDUT
(*
SPDX-FileCopyrightText: © 2026 Oleksandr Tiutyk <trofimich@gmail.com>
SPDX-License-Identifier: MIT
License: https://opensource.org/license/mit
*)

(*!
<summary>
Beckhoff EL1008: 8-channel digital input terminal (24 V DC, 3 ms filter).
</summary>
<description>
Process image mapping structure for the EL1008 standard 8-channel discrete 24 V DC input terminal.
When used for I/O, link located fields or their containing buffers to the matching selected PDOs.
The record is not a packed wire buffer; compiler padding is not part of the device specification.
Unlinked/default values do not prove valid I/O. The caller evaluates bus/channel validity before use.
Use one owner task per instance and externally synchronize other access; multi-field snapshots are not atomic.
Copies store data without creating hardware links. Keep borrowed field references valid while consumers are bound.
This passive record performs no validation, synchronization, configuration or protocol advancement.
</description>
*)
TYPE EL1008 :
STRUCT
	Ch1 AT %I* : BOOL;
	Ch2 AT %I* : BOOL;
	Ch3 AT %I* : BOOL;
	Ch4 AT %I* : BOOL;
	Ch5 AT %I* : BOOL;
	Ch6 AT %I* : BOOL;
	Ch7 AT %I* : BOOL;
	Ch8 AT %I* : BOOL;
END_STRUCT
END_TYPE

// ---- DigitalIO/Inputs/EL1008/EL1008_EX.TcDUT
(*
SPDX-FileCopyrightText: © 2026 Oleksandr Tiutyk <trofimich@gmail.com>
SPDX-License-Identifier: MIT
License: https://opensource.org/license/mit
*)

